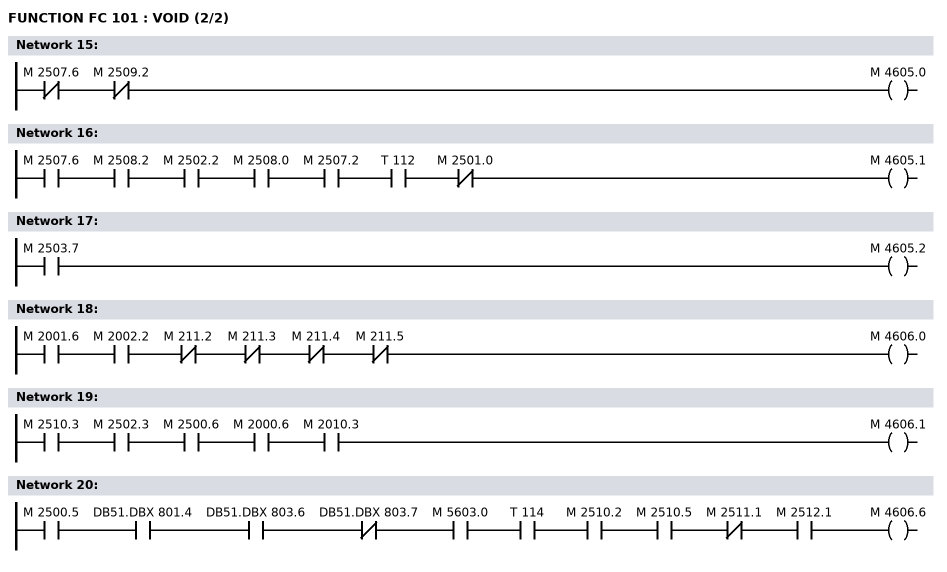

      AN    M   2507.6;
      AN    M   2509.2;
      =     M   4605.0;
NETWORK
TITLE =

      A     M   2507.6;
      A     M   2508.2;
      A     M   2502.2;
      A     M   2508.0;
      A     M   2507.2;
      A     T    112;
      AN    M   2501.0;
      =     M   4605.1;
NETWORK
TITLE =

      A     M   2503.7;
      =     M   4605.2;
NETWORK
TITLE =

      A     M   2001.6;
      A     M   2002.2;
      AN    M    211.2;
      AN    M    211.3;
      AN    M    211.4;
      AN    M    211.5;
      =     M   4606.0;
NETWORK
TITLE =

      A     M   2510.3;
      A     M   2502.3;
      A     M   2500.6;
      A     M   2000.6;
      A     M   2010.3;
      =     M   4606.1;
NETWORK
TITLE =

      A     M   2500.5;
      A     DB51.DBX  801.4;
      A     DB51.DBX  803.6;
      AN    DB51.DBX  803.7;
      A     M   5603.0;
      A     T    114;
      A     M   2510.2;
      A     M   2510.5;
      AN    M   2511.1;
      A     M   2512.1;
      =     M   4606.6;
END_FUNCTION

FUNCTION FC 102 : VOID
TITLE =
VERSION : 0.1

BEGIN
NETWORK
TITLE =운전준비
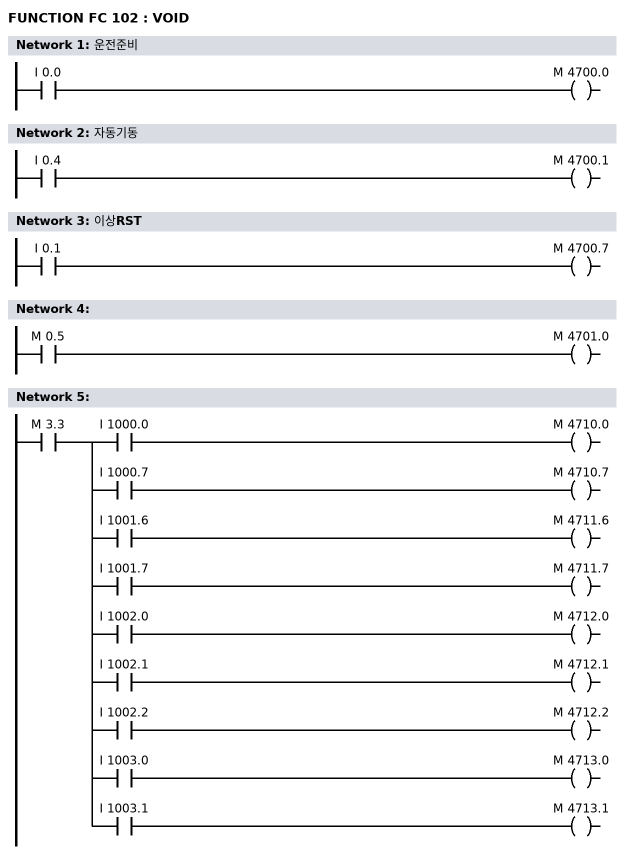

      A     I      0.0;
      =     M   4700.0;
NETWORK
TITLE =자동기동

      A     I      0.4;
      =     M   4700.1;
NETWORK
TITLE =이상RST

      A     I      0.1;
      =     M   4700.7;
NETWORK
TITLE =

      A     M      0.5;
      =     M   4701.0;
NETWORK
TITLE =

      A     M      3.3;
      =     L      0.0;
      A     L      0.0;
      A     I   1000.0;
      =     M   4710.0;
      A     L      0.0;
      A     I   1000.7;
      =     M   4710.7;
      A     L      0.0;
      A     I   1001.6;
      =     M   4711.6;
      A     L      0.0;
      A     I   1001.7;
      =     M   4711.7;
      A     L      0.0;
      A     I   1002.0;
      =     M   4712.0;
      A     L      0.0;
      A     I   1002.1;
      =     M   4712.1;
      A     L      0.0;
      A     I   1002.2;
      =     M   4712.2;
      A     L      0.0;
      A     I   1003.0;
      =     M   4713.0;
      A     L      0.0;
      A     I   1003.1;
      =     M   4713.1;
END_FUNCTION

FUNCTION FC 103 : VOID
TITLE =
VERSION : 0.1

BEGIN
NETWORK
TITLE =
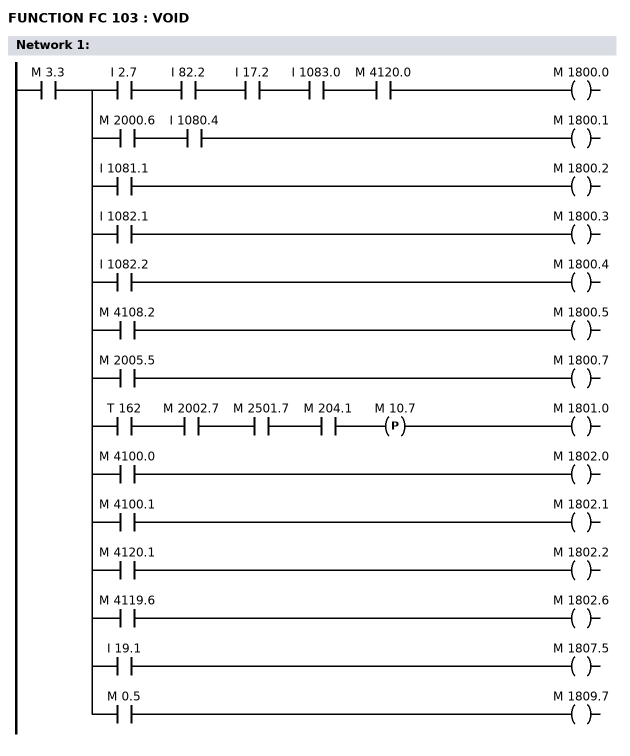

      A     M      3.3;
      =     L      0.0;
      A     L      0.0;
      A     I      2.7;
      A     I     82.2;
      A     I     17.2;
      A     I   1083.0;
      A     M   4120.0;
      =     M   1800.0;
      A     L      0.0;
      A     M   2000.6;
      A     I   1080.4;
      =     M   1800.1;
      A     L      0.0;
      A     I   1081.1;
      =     M   1800.2;
      A     L      0.0;
      A     I   1082.1;
      =     M   1800.3;
      A     L      0.0;
      A     I   1082.2;
      =     M   1800.4;
      A     L      0.0;
      A     M   4108.2;
      =     M   1800.5;
      A     L      0.0;
      A     M   2005.5;
      =     M   1800.7;
      A     L      0.0;
      A     T    162;
      A     M   2002.7;
      A     M   2501.7;
      A     M    204.1;
      FP    M     10.7;
      =     M   1801.0;
      A     L      0.0;
      A     M   4100.0;
      =     M   1802.0;
      A     L      0.0;
      A     M   4100.1;
      =     M   1802.1;
      A     L      0.0;
      A     M   4120.1;
      =     M   1802.2;
      A     L      0.0;
      A     M   4119.6;
      =     M   1802.6;
      A     L      0.0;
      A     I     19.1;
      =     M   1807.5;
      A     L      0.0;
      A     M      0.5;
      =     M   1809.7;
END_FUNCTION

FUNCTION_BLOCK FB 105
TITLE =
VERSION : 0.1


VAR
  S705_RBT1_WELD_OK_PLS : BOOL ;
  S705_RBT1_WELD_NG_PLS : BOOL ;
  S705_RBT1_WELD_PASS_PLS : BOOL ;
  S705_CHECK_SUM_PLS : BOOL ;
  S705_WELD_DATA_MOV_BUFF : BOOL ;
  MW_0_BUFF : ARRAY  [0 .. 59 ] OF WORD ;
  S706_RBT1_WELD_OK_PLS : BOOL ;
  S706_RBT1_WELD_NG_PLS : BOOL ;
  S706_RBT1_WELD_PASS_PLS : BOOL ;
  S706_RBT2_WELD_OK_PLS : BOOL ;
  S706_RBT2_WELD_NG_PLS : BOOL ;
  S706_RBT2_WELD_PASS_PLS : BOOL ;
  S706_RBT3_WELD_OK_PLS : BOOL ;
  S706_RBT3_WELD_NG_PLS : BOOL ;
  S706_RBT3_WELD_PASS_PLS : BOOL ;
  S706_CHECK_SUM_PLS : BOOL ;
  S706_WELD_DATA_MOV_BUFF : BOOL ;
  S711_RBT1_WELD_OK_PLS : BOOL ;
  S711_RBT1_WELD_NG_PLS : BOOL ;
  S711_RBT1_WELD_PASS_PLS : BOOL ;
  S711_CHECK_SUM_PLS : BOOL ;
  S711_WELD_DATA_MOV_BUFF : BOOL ;
  PLS1 : BOOL ;
  PLS2 : BOOL ;
  PLS3 : BOOL ;
  PLS4 : BOOL ;
  PLS5 : BOOL ;
  PLS6 : BOOL ;
END_VAR
VAR_TEMP
  SFC20_RET_VAL : INT ;
END_VAR
BEGIN
NETWORK
TITLE =MES 용접누락 DATA -> #705차종코드(2011) 기준값 버퍼로 전송(LM)
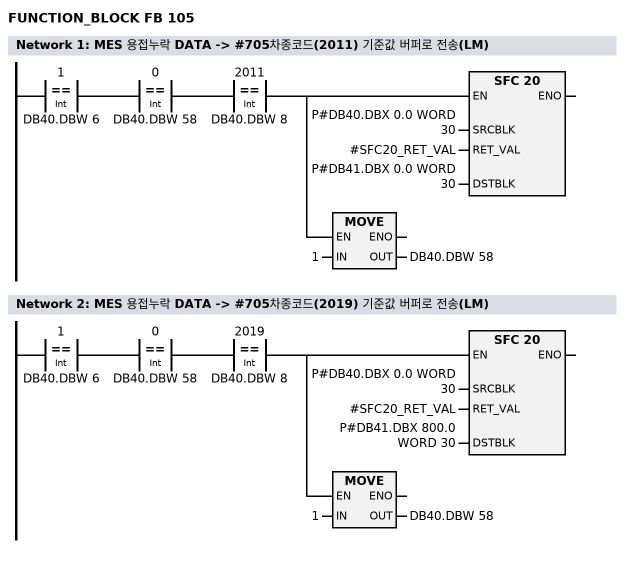

      A(    ;
      L     1;
      L     DB40.DBW    6;
      ==I   ;
      )     ;
      A(    ;
      L     0;
      L     DB40.DBW   58;
      ==I   ;
      )     ;
      A(    ;
      L     2011;
      L     DB40.DBW    8;
      ==I   ;
      )     ;
      =     L      2.0;
      A     L      2.0;
      JNB   _001;
      CALL SFC   20 (
           SRCBLK                   := P#DB40.DBX 0.0 WORD 30,
           RET_VAL                  := #SFC20_RET_VAL,
           DSTBLK                   := P#DB41.DBX 0.0 WORD 30);
_001: NOP   0;
      A     L      2.0;
      JNB   _002;
      L     1;
      T     DB40.DBW   58;
_002: NOP   0;
NETWORK
TITLE =MES 용접누락 DATA -> #705차종코드(2019) 기준값 버퍼로 전송(LM)

      A(    ;
      L     1;
      L     DB40.DBW    6;
      ==I   ;
      )     ;
      A(    ;
      L     0;
      L     DB40.DBW   58;
      ==I   ;
      )     ;
      A(    ;
      L     2019;
      L     DB40.DBW    8;
      ==I   ;
      )     ;
      =     L      2.0;
      A     L      2.0;
      JNB   _003;
      CALL SFC   20 (
           SRCBLK                   := P#DB40.DBX 0.0 WORD 30,
           RET_VAL                  := #SFC20_RET_VAL,
           DSTBLK                   := P#DB41.DBX 800.0 WORD 30);
_003: NOP   0;
      A     L      2.0;
      JNB   _004;
      L     1;
      T     DB40.DBW   58;
_004: NOP   0;
NETWORK
TITLE =#705 RBT1호 용접카운터 INT -> DB로 전송보조

      AN    OV;
      =     L      2.0;
      A     L      2.0;
      A     I   1004.0;
      =     M     11.0;
      A     L      2.0;
      A     I   1004.1;
      =     M     11.1;
      A     L      2.0;
      A     I   1004.2;
      =     M     11.2;
      A     L      2.0;
      A     I   1004.3;
      =     M     11.3;
      A     L      2.0;
      A     I   1004.4;
      =     M     11.4;
      A     L      2.0;
      AN    M      3.3;
      =     L      2.1;
      A     L      2.1;
      A     I   1004.5;
      =     M     11.5;
      A     L      2.1;
      A     I   1004.6;
      =     M     11.6;
      A     L      2.1;
      A     I   1004.7;
      =     M     11.7;
NETWORK
TITLE =#705 RBT1호 용접카운터 INT -> DB로 전송
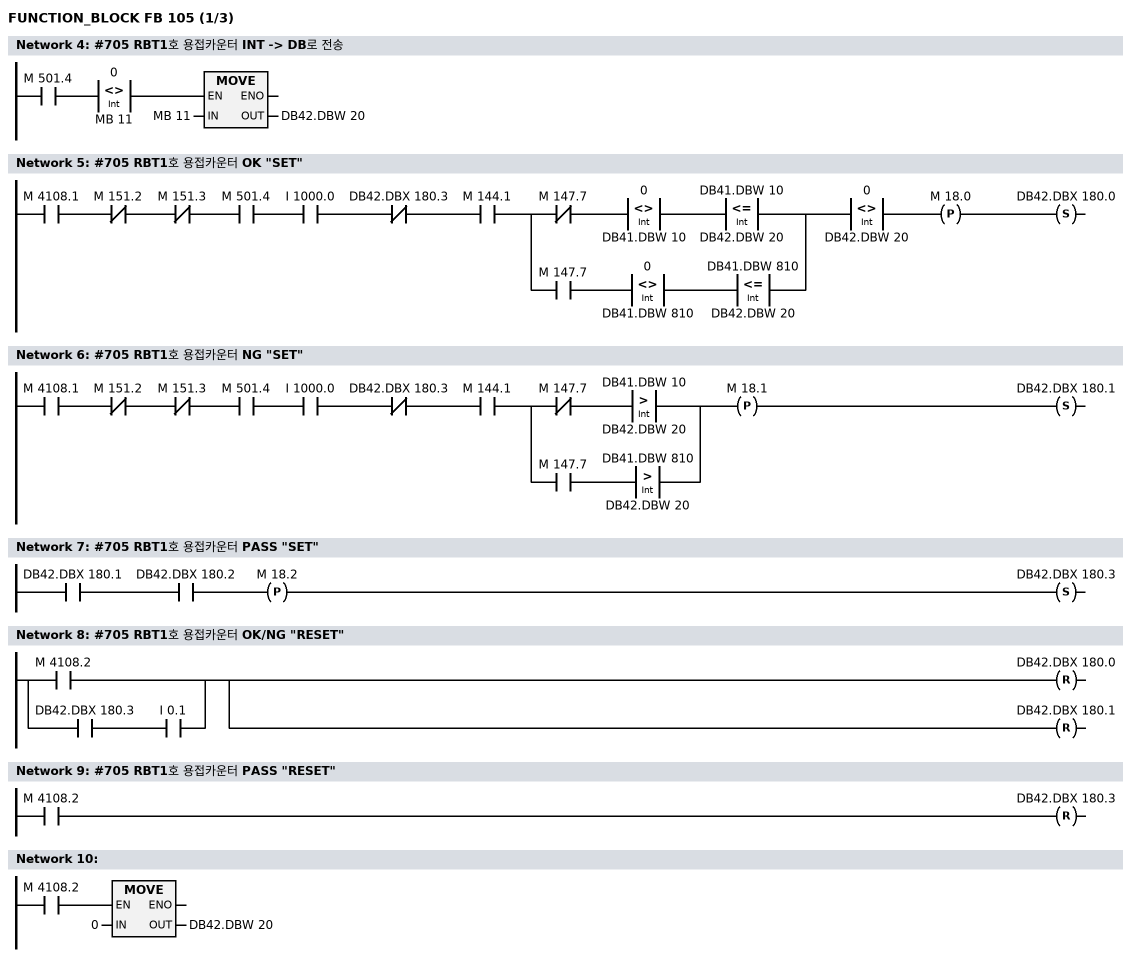

      A     M    501.4;
      A(    ;
      L     0;
      L     MB    11;
      <>I   ;
      )     ;
      JNB   _005;
      L     MB    11;
      T     DB42.DBW   20;
_005: NOP   0;
NETWORK
TITLE =#705 RBT1호 용접카운터 OK "SET"

      A     M   4108.1;
      AN    M    151.2;
      AN    M    151.3;
      A     M    501.4;
      A     I   1000.0;
      AN    DB42.DBX  180.3;
      A     M    144.1;
      A(    ;
      AN    M    147.7;
      A(    ;
      L     0;
      L     DB41.DBW   10;
      <>I   ;
      )     ;
      A(    ;
      L     DB41.DBW   10;
      L     DB42.DBW   20;
      <=I   ;
      )     ;
      O     ;
      A     M    147.7;
      A(    ;
      L     0;
      L     DB41.DBW  810;
      <>I   ;
      )     ;
      A(    ;
      L     DB41.DBW  810;
      L     DB42.DBW   20;
      <=I   ;
      )     ;
      )     ;
      A(    ;
      L     0;
      L     DB42.DBW   20;
      <>I   ;
      )     ;
      FP    M     18.0;
      S     DB42.DBX  180.0;
NETWORK
TITLE =#705 RBT1호 용접카운터 NG "SET"

      A     M   4108.1;
      AN    M    151.2;
      AN    M    151.3;
      A     M    501.4;
      A     I   1000.0;
      AN    DB42.DBX  180.3;
      A     M    144.1;
      A(    ;
      AN    M    147.7;
      A(    ;
      L     DB41.DBW   10;
      L     DB42.DBW   20;
      >I    ;
      )     ;
      O     ;
      A     M    147.7;
      A(    ;
      L     DB41.DBW  810;
      L     DB42.DBW   20;
      >I    ;
      )     ;
      )     ;
      FP    M     18.1;
      S     DB42.DBX  180.1;
NETWORK
TITLE =#705 RBT1호 용접카운터 PASS "SET"

      A     DB42.DBX  180.1;
      A     DB42.DBX  180.2;
      FP    M     18.2;
      S     DB42.DBX  180.3;
NETWORK
TITLE =#705 RBT1호 용접카운터 OK/NG "RESET"

      O     M   4108.2;
      O     ;
      A     DB42.DBX  180.3;
      A     I      0.1;
      R     DB42.DBX  180.0;
      R     DB42.DBX  180.1;
NETWORK
TITLE =#705 RBT1호 용접카운터 PASS "RESET"

      A     M   4108.2;
      R     DB42.DBX  180.3;
NETWORK
TITLE =

      A     M   4108.2;
      JNB   _006;
      L     0;
      T     DB42.DBW   20;
_006: NOP   0;
NETWORK
TITLE =
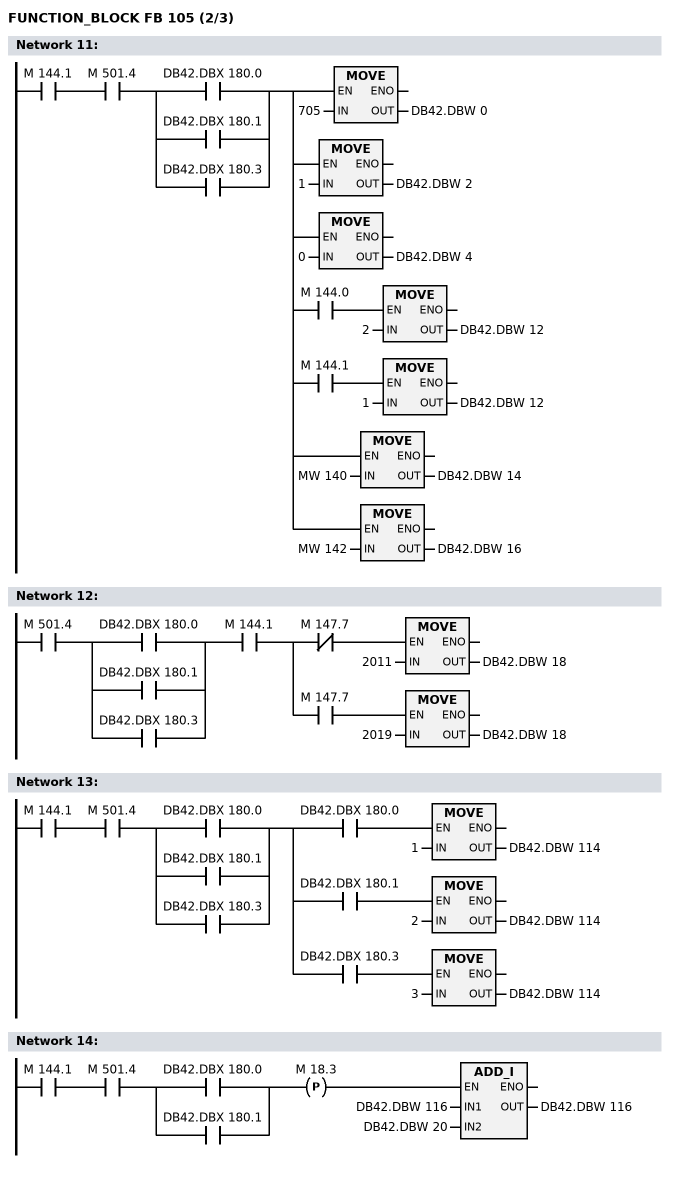

      A     M    144.1;
      A     M    501.4;
      A(    ;
      O     DB42.DBX  180.0;
      O     DB42.DBX  180.1;
      O     DB42.DBX  180.3;
      )     ;
      =     L      2.0;
      A     L      2.0;
      JNB   _007;
      L     705;
      T     DB42.DBW    0;
_007: NOP   0;
      A     L      2.0;
      JNB   _008;
      L     1;
      T     DB42.DBW    2;
_008: NOP   0;
      A     L      2.0;
      JNB   _009;
      L     0;
      T     DB42.DBW    4;
_009: NOP   0;
      A     L      2.0;
      A     M    144.0;
      JNB   _00a;
      L     2;
      T     DB42.DBW   12;
_00a: NOP   0;
      A     L      2.0;
      A     M    144.1;
      JNB   _00b;
      L     1;
      T     DB42.DBW   12;
_00b: NOP   0;
      A     L      2.0;
      JNB   _00c;
      L     MW   140;
      T     DB42.DBW   14;
_00c: NOP   0;
      A     L      2.0;
      JNB   _00d;
      L     MW   142;
      T     DB42.DBW   16;
_00d: NOP   0;
NETWORK
TITLE =

      A     M    501.4;
      A(    ;
      O     DB42.DBX  180.0;
      O     DB42.DBX  180.1;
      O     DB42.DBX  180.3;
      )     ;
      A     M    144.1;
      =     L      2.0;
      A     L      2.0;
      AN    M    147.7;
      JNB   _00e;
      L     2011;
      T     DB42.DBW   18;
_00e: NOP   0;
      A     L      2.0;
      A     M    147.7;
      JNB   _00f;
      L     2019;
      T     DB42.DBW   18;
_00f: NOP   0;
NETWORK
TITLE =

      A     M    144.1;
      A     M    501.4;
      A(    ;
      O     DB42.DBX  180.0;
      O     DB42.DBX  180.1;
      O     DB42.DBX  180.3;
      )     ;
      =     L      2.0;
      A     L      2.0;
      A     DB42.DBX  180.0;
      JNB   _010;
      L     1;
      T     DB42.DBW  114;
_010: NOP   0;
      A     L      2.0;
      A     DB42.DBX  180.1;
      JNB   _011;
      L     2;
      T     DB42.DBW  114;
_011: NOP   0;
      A     L      2.0;
      A     DB42.DBX  180.3;
      JNB   _012;
      L     3;
      T     DB42.DBW  114;
_012: NOP   0;
NETWORK
TITLE =

      A     M    144.1;
      A     M    501.4;
      A(    ;
      O     DB42.DBX  180.0;
      O     DB42.DBX  180.1;
      )     ;
      FP    M     18.3;
      JNB   _013;
      L     DB42.DBW  116;
      L     DB42.DBW   20;
      +I    ;
      T     DB42.DBW  116;
_013: NOP   0;
NETWORK
TITLE =
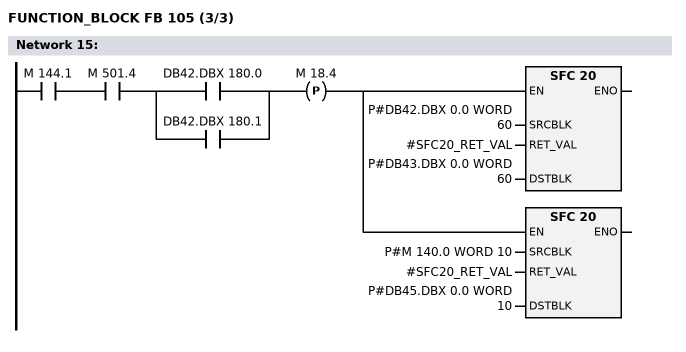

      A     M    144.1;
      A     M    501.4;
      A(    ;
      O     DB42.DBX  180.0;
      O     DB42.DBX  180.1;
      )     ;
      FP    M     18.4;
      =     L      2.0;
      A     L      2.0;
      JNB   _014;
      CALL SFC   20 (
           SRCBLK                   := P#DB42.DBX 0.0 WORD 60,
           RET_VAL                  := #SFC20_RET_VAL,
           DSTBLK                   := P#DB43.DBX 0.0 WORD 60);
_014: NOP   0;
      A     L      2.0;
      JNB   _015;
      CALL SFC   20 (
           SRCBLK                   := P#M 140.0 WORD 10,
           RET_VAL                  := #SFC20_RET_VAL,
           DSTBLK                   := P#DB45.DBX 0.0 WORD 10);
_015: NOP   0;
NETWORK
TITLE =

      A     M   4108.2;
      FP    M     18.5;
      =     L      2.0;
      A(    ;
      A     L      2.0;
      JNB   _016;
      CALL SFC   20 (
           SRCBLK                   := P#DB43.DBX 960.0 WORD 60,
           RET_VAL                  := #SFC20_RET_VAL,
           DSTBLK                   := P#DB43.DBX 1080.0 WORD 60);
_016: A     BR;
      )     ;
      JNB   _017;
      CALL SFC   20 (
           SRCBLK                   := P#DB43.DBX 840.0 WORD 60,
           RET_VAL                  := #SFC20_RET_VAL,
           DSTBLK                   := P#DB43.DBX 960.0 WORD 60);
_017: NOP   0;
      A(    ;
      A     L      2.0;
      JNB   _018;
      CALL SFC   20 (
           SRCBLK                   := P#DB43.DBX 720.0 WORD 60,
           RET_VAL                  := #SFC20_RET_VAL,
           DSTBLK                   := P#DB43.DBX 840.0 WORD 60);
_018: A     BR;
      )     ;
      JNB   _019;
      CALL SFC   20 (
           SRCBLK                   := P#DB43.DBX 600.0 WORD 60,
           RET_VAL                  := #SFC20_RET_VAL,
           DSTBLK                   := P#DB43.DBX 720.0 WORD 60);
_019: NOP   0;
      A(    ;
      A     L      2.0;
      JNB   _01a;
      CALL SFC   20 (
           SRCBLK                   := P#DB43.DBX 480.0 WORD 60,
           RET_VAL                  := #SFC20_RET_VAL,
           DSTBLK                   := P#DB43.DBX 600.0 WORD 60);
_01a: A     BR;
      )     ;
      JNB   _01b;
      CALL SFC   20 (
           SRCBLK                   := P#DB43.DBX 360.0 WORD 60,
           RET_VAL                  := #SFC20_RET_VAL,
           DSTBLK                   := P#DB43.DBX 480.0 WORD 60);
_01b: NOP   0;
      A(    ;
      A     L      2.0;
      JNB   _01c;
      CALL SFC   20 (
           SRCBLK                   := P#DB43.DBX 240.0 WORD 60,
           RET_VAL                  := #SFC20_RET_VAL,
           DSTBLK                   := P#DB43.DBX 360.0 WORD 60);
_01c: A     BR;
      )     ;
      JNB   _01d;
      CALL SFC   20 (
           SRCBLK                   := P#DB43.DBX 120.0 WORD 60,
           RET_VAL                  := #SFC20_RET_VAL,
           DSTBLK                   := P#DB43.DBX 240.0 WORD 60);
_01d: NOP   0;
      A     L      2.0;
      JNB   _01e;
      CALL SFC   20 (
           SRCBLK                   := P#DB43.DBX 0.0 WORD 60,
           RET_VAL                  := #SFC20_RET_VAL,
           DSTBLK                   := P#DB43.DBX 120.0 WORD 60);
_01e: NOP   0;
      A     L      2.0;
      JNB   _01f;
      CALL SFC   21 (
           IN0                      := P#M 40.0 WORD 1,
           RET_VAL                  := #SFC20_RET_VAL,
           OUT1                     := P#DB43.DBX 0.0 WORD 60);
_01f: NOP   0;
      A(    ;
      A     L      2.0;
      JNB   _020;
      CALL SFC   20 (
           SRCBLK                   := P#DB45.DBX 160.0 WORD 10,
           RET_VAL                  := #SFC20_RET_VAL,
           DSTBLK                   := P#DB45.DBX 180.0 WORD 10);
_020: A     BR;
      )     ;
      JNB   _021;
      CALL SFC   20 (
           SRCBLK                   := P#DB45.DBX 140.0 WORD 10,
           RET_VAL                  := #SFC20_RET_VAL,
           DSTBLK                   := P#DB45.DBX 160.0 WORD 10);
_021: NOP   0;
      A(    ;
      A     L      2.0;
      JNB   _022;
      CALL SFC   20 (
           SRCBLK                   := P#DB45.DBX 120.0 WORD 10,
           RET_VAL                  := #SFC20_RET_VAL,
           DSTBLK                   := P#DB45.DBX 140.0 WORD 10);
_022: A     BR;
      )     ;
      JNB   _023;
      CALL SFC   20 (
           SRCBLK                   := P#DB45.DBX 100.0 WORD 10,
           RET_VAL                  := #SFC20_RET_VAL,
           DSTBLK                   := P#DB45.DBX 120.0 WORD 10);
_023: NOP   0;
      A(    ;
      A     L      2.0;
      JNB   _024;
      CALL SFC   20 (
           SRCBLK                   := P#DB45.DBX 80.0 WORD 10,
           RET_VAL                  := #SFC20_RET_VAL,
           DSTBLK                   := P#DB45.DBX 100.0 WORD 10);
_024: A     BR;
      )     ;
      JNB   _025;
      CALL SFC   20 (
           SRCBLK                   := P#DB45.DBX 60.0 WORD 10,
           RET_VAL                  := #SFC20_RET_VAL,
           DSTBLK                   := P#DB45.DBX 80.0 WORD 10);
_025: NOP   0;
      A(    ;
      A     L      2.0;
      JNB   _026;
      CALL SFC   20 (
           SRCBLK                   := P#DB45.DBX 40.0 WORD 10,
           RET_VAL                  := #SFC20_RET_VAL,
           DSTBLK                   := P#DB45.DBX 60.0 WORD 10);
_026: A     BR;
      )     ;
      JNB   _027;
      CALL SFC   20 (
           SRCBLK                   := P#DB45.DBX 20.0 WORD 10,
           RET_VAL                  := #SFC20_RET_VAL,
           DSTBLK                   := P#DB45.DBX 40.0 WORD 10);
_027: NOP   0;
      A     L      2.0;
      JNB   _028;
      CALL SFC   20 (
           SRCBLK                   := P#DB45.DBX 0.0 WORD 10,
           RET_VAL                  := #SFC20_RET_VAL,
           DSTBLK                   := P#DB45.DBX 20.0 WORD 10);
_028: NOP   0;
      A     L      2.0;
      JNB   _029;
      CALL SFC   21 (
           IN0                      := P#M 40.0 WORD 1,
           RET_VAL                  := #SFC20_RET_VAL,
           OUT1                     := P#DB45.DBX 0.0 WORD 10);
_029: NOP   0;
NETWORK
TITLE =
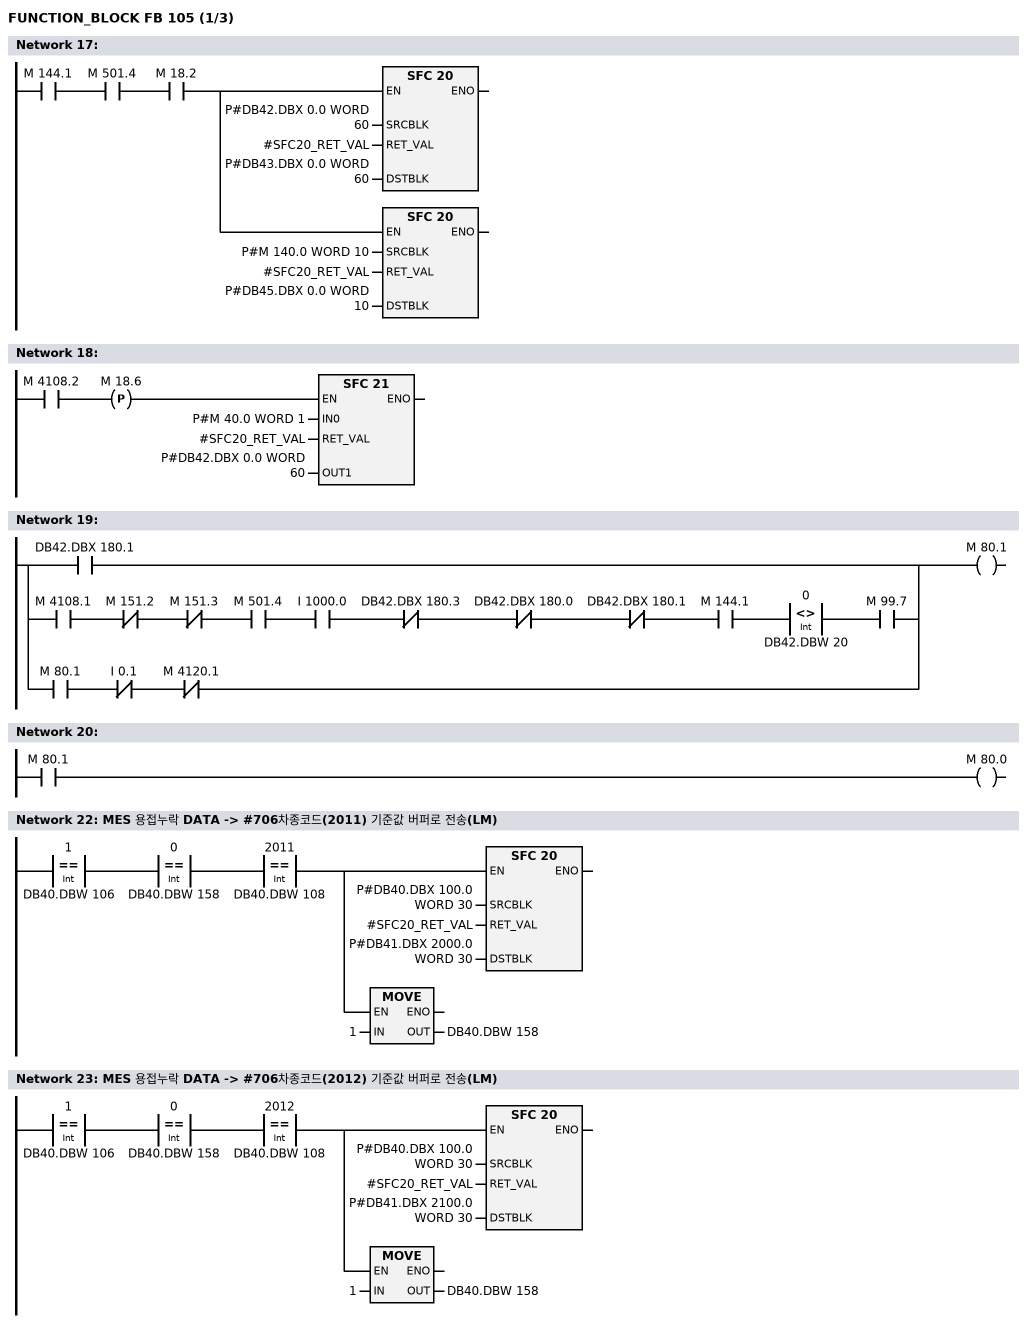

      A     M    144.1;
      A     M    501.4;
      A     M     18.2;
      =     L      2.0;
      A     L      2.0;
      JNB   _02a;
      CALL SFC   20 (
           SRCBLK                   := P#DB42.DBX 0.0 WORD 60,
           RET_VAL                  := #SFC20_RET_VAL,
           DSTBLK                   := P#DB43.DBX 0.0 WORD 60);
_02a: NOP   0;
      A     L      2.0;
      JNB   _02b;
      CALL SFC   20 (
           SRCBLK                   := P#M 140.0 WORD 10,
           RET_VAL                  := #SFC20_RET_VAL,
           DSTBLK                   := P#DB45.DBX 0.0 WORD 10);
_02b: NOP   0;
NETWORK
TITLE =

      A     M   4108.2;
      FP    M     18.6;
      JNB   _02c;
      CALL SFC   21 (
           IN0                      := P#M 40.0 WORD 1,
           RET_VAL                  := #SFC20_RET_VAL,
           OUT1                     := P#DB42.DBX 0.0 WORD 60);
_02c: NOP   0;
NETWORK
TITLE =

      O     DB42.DBX  180.1;
      O     ;
      A     M   4108.1;
      AN    M    151.2;
      AN    M    151.3;
      A     M    501.4;
      A     I   1000.0;
      AN    DB42.DBX  180.3;
      AN    DB42.DBX  180.0;
      AN    DB42.DBX  180.1;
      A     M    144.1;
      A(    ;
      L     0;
      L     DB42.DBW   20;
      <>I   ;
      )     ;
      A     M     99.7;
      O     ;
      A     M     80.1;
      AN    I      0.1;
      AN    M   4120.1;
      =     M     80.1;
NETWORK
TITLE =

      A     M     80.1;
      =     M     80.0;
NETWORK
TITLE =

NETWORK
TITLE =MES 용접누락 DATA -> #706차종코드(2011) 기준값 버퍼로 전송(LM)

      A(    ;
      L     1;
      L     DB40.DBW  106;
      ==I   ;
      )     ;
      A(    ;
      L     0;
      L     DB40.DBW  158;
      ==I   ;
      )     ;
      A(    ;
      L     2011;
      L     DB40.DBW  108;
      ==I   ;
      )     ;
      =     L      2.0;
      A     L      2.0;
      JNB   _02d;
      CALL SFC   20 (
           SRCBLK                   := P#DB40.DBX 100.0 WORD 30,
           RET_VAL                  := #SFC20_RET_VAL,
           DSTBLK                   := P#DB41.DBX 2000.0 WORD 30);
_02d: NOP   0;
      A     L      2.0;
      JNB   _02e;
      L     1;
      T     DB40.DBW  158;
_02e: NOP   0;
NETWORK
TITLE =MES 용접누락 DATA -> #706차종코드(2012) 기준값 버퍼로 전송(LM)

      A(    ;
      L     1;
      L     DB40.DBW  106;
      ==I   ;
      )     ;
      A(    ;
      L     0;
      L     DB40.DBW  158;
      ==I   ;
      )     ;
      A(    ;
      L     2012;
      L     DB40.DBW  108;
      ==I   ;
      )     ;
      =     L      2.0;
      A     L      2.0;
      JNB   _02f;
      CALL SFC   20 (
           SRCBLK                   := P#DB40.DBX 100.0 WORD 30,
           RET_VAL                  := #SFC20_RET_VAL,
           DSTBLK                   := P#DB41.DBX 2100.0 WORD 30);
_02f: NOP   0;
      A     L      2.0;
      JNB   _030;
      L     1;
      T     DB40.DBW  158;
_030: NOP   0;
NETWORK
TITLE =MES 용접누락 DATA -> #706차종코드(2013) 기준값 버퍼로 전송(LM)
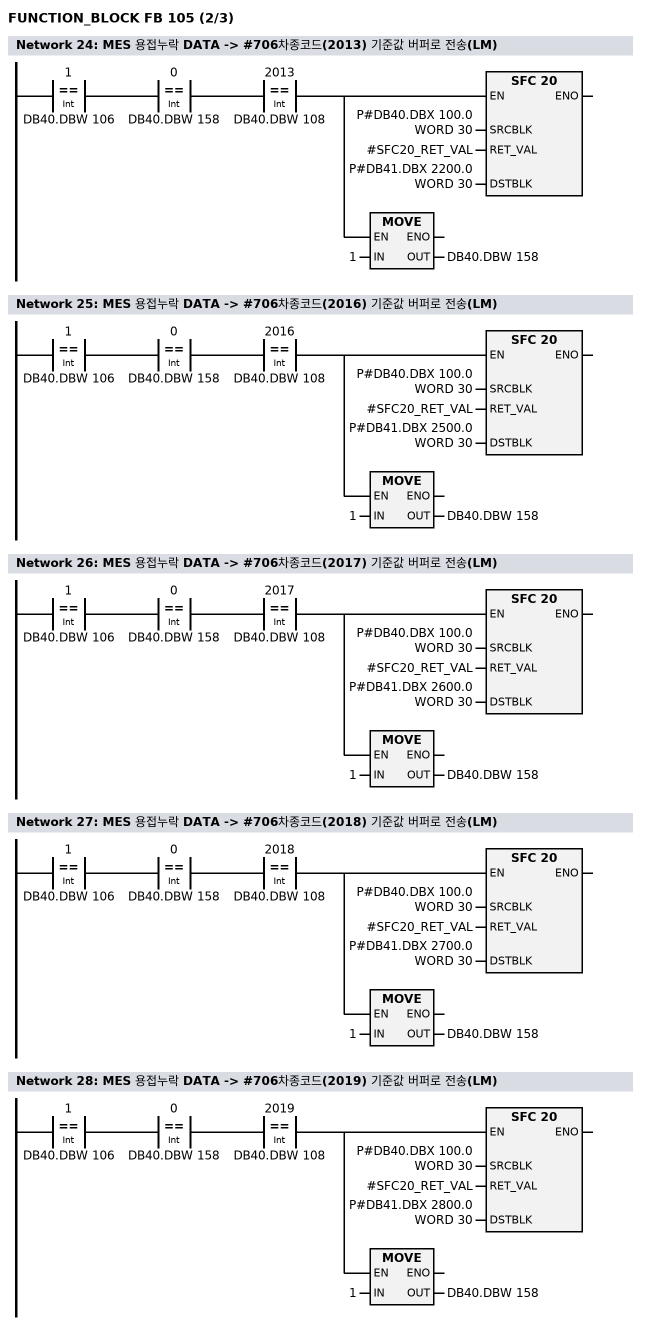

      A(    ;
      L     1;
      L     DB40.DBW  106;
      ==I   ;
      )     ;
      A(    ;
      L     0;
      L     DB40.DBW  158;
      ==I   ;
      )     ;
      A(    ;
      L     2013;
      L     DB40.DBW  108;
      ==I   ;
      )     ;
      =     L      2.0;
      A     L      2.0;
      JNB   _031;
      CALL SFC   20 (
           SRCBLK                   := P#DB40.DBX 100.0 WORD 30,
           RET_VAL                  := #SFC20_RET_VAL,
           DSTBLK                   := P#DB41.DBX 2200.0 WORD 30);
_031: NOP   0;
      A     L      2.0;
      JNB   _032;
      L     1;
      T     DB40.DBW  158;
_032: NOP   0;
NETWORK
TITLE =MES 용접누락 DATA -> #706차종코드(2016) 기준값 버퍼로 전송(LM)

      A(    ;
      L     1;
      L     DB40.DBW  106;
      ==I   ;
      )     ;
      A(    ;
      L     0;
      L     DB40.DBW  158;
      ==I   ;
      )     ;
      A(    ;
      L     2016;
      L     DB40.DBW  108;
      ==I   ;
      )     ;
      =     L      2.0;
      A     L      2.0;
      JNB   _033;
      CALL SFC   20 (
           SRCBLK                   := P#DB40.DBX 100.0 WORD 30,
           RET_VAL                  := #SFC20_RET_VAL,
           DSTBLK                   := P#DB41.DBX 2500.0 WORD 30);
_033: NOP   0;
      A     L      2.0;
      JNB   _034;
      L     1;
      T     DB40.DBW  158;
_034: NOP   0;
NETWORK
TITLE =MES 용접누락 DATA -> #706차종코드(2017) 기준값 버퍼로 전송(LM)

      A(    ;
      L     1;
      L     DB40.DBW  106;
      ==I   ;
      )     ;
      A(    ;
      L     0;
      L     DB40.DBW  158;
      ==I   ;
      )     ;
      A(    ;
      L     2017;
      L     DB40.DBW  108;
      ==I   ;
      )     ;
      =     L      2.0;
      A     L      2.0;
      JNB   _035;
      CALL SFC   20 (
           SRCBLK                   := P#DB40.DBX 100.0 WORD 30,
           RET_VAL                  := #SFC20_RET_VAL,
           DSTBLK                   := P#DB41.DBX 2600.0 WORD 30);
_035: NOP   0;
      A     L      2.0;
      JNB   _036;
      L     1;
      T     DB40.DBW  158;
_036: NOP   0;
NETWORK
TITLE =MES 용접누락 DATA -> #706차종코드(2018) 기준값 버퍼로 전송(LM)

      A(    ;
      L     1;
      L     DB40.DBW  106;
      ==I   ;
      )     ;
      A(    ;
      L     0;
      L     DB40.DBW  158;
      ==I   ;
      )     ;
      A(    ;
      L     2018;
      L     DB40.DBW  108;
      ==I   ;
      )     ;
      =     L      2.0;
      A     L      2.0;
      JNB   _037;
      CALL SFC   20 (
           SRCBLK                   := P#DB40.DBX 100.0 WORD 30,
           RET_VAL                  := #SFC20_RET_VAL,
           DSTBLK                   := P#DB41.DBX 2700.0 WORD 30);
_037: NOP   0;
      A     L      2.0;
      JNB   _038;
      L     1;
      T     DB40.DBW  158;
_038: NOP   0;
NETWORK
TITLE =MES 용접누락 DATA -> #706차종코드(2019) 기준값 버퍼로 전송(LM)

      A(    ;
      L     1;
      L     DB40.DBW  106;
      ==I   ;
      )     ;
      A(    ;
      L     0;
      L     DB40.DBW  158;
      ==I   ;
      )     ;
      A(    ;
      L     2019;
      L     DB40.DBW  108;
      ==I   ;
      )     ;
      =     L      2.0;
      A     L      2.0;
      JNB   _039;
      CALL SFC   20 (
           SRCBLK                   := P#DB40.DBX 100.0 WORD 30,
           RET_VAL                  := #SFC20_RET_VAL,
           DSTBLK                   := P#DB41.DBX 2800.0 WORD 30);
_039: NOP   0;
      A     L      2.0;
      JNB   _03a;
      L     1;
      T     DB40.DBW  158;
_03a: NOP   0;
NETWORK
TITLE =MES 용접누락 DATA -> #706차종코드(2101) 기준값 버퍼로 전송(TL)
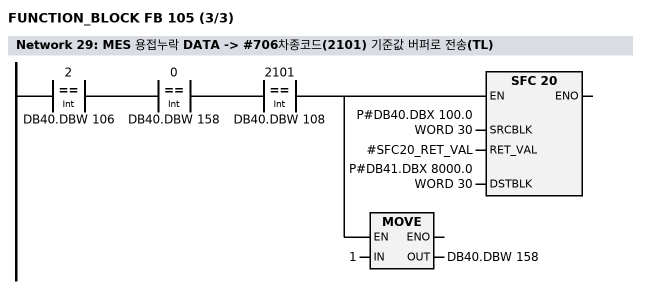

      A(    ;
      L     2;
      L     DB40.DBW  106;
      ==I   ;
      )     ;
      A(    ;
      L     0;
      L     DB40.DBW  158;
      ==I   ;
      )     ;
      A(    ;
      L     2101;
      L     DB40.DBW  108;
      ==I   ;
      )     ;
      =     L      2.0;
      A     L      2.0;
      JNB   _03b;
      CALL SFC   20 (
           SRCBLK                   := P#DB40.DBX 100.0 WORD 30,
           RET_VAL                  := #SFC20_RET_VAL,
           DSTBLK                   := P#DB41.DBX 8000.0 WORD 30);
_03b: NOP   0;
      A     L      2.0;
      JNB   _03c;
      L     1;
      T     DB40.DBW  158;
_03c: NOP   0;
NETWORK
TITLE =#706 RBT1호 용접카운터 INT -> DB로 전송보조

      AN    OV;
      =     L      2.0;
      A     L      2.0;
      A     I   1028.0;
      =     M     12.0;
      A     L      2.0;
      A     I   1028.1;
      =     M     12.1;
      A     L      2.0;
      A     I   1028.2;
      =     M     12.2;
      A     L      2.0;
      A     I   1028.3;
      =     M     12.3;
      A     L      2.0;
      A     I   1028.4;
      =     M     12.4;
      A     L      2.0;
      AN    M      3.3;
      =     L      2.1;
      A     L      2.1;
      A     I   1028.5;
      =     M     12.5;
      A     L      2.1;
      A     I   1028.6;
      =     M     12.6;
      A     L      2.1;
      A     I   1028.7;
      =     M     12.7;
NETWORK
TITLE =#706 RBT1호 용접카운터 INT -> DB로 전송
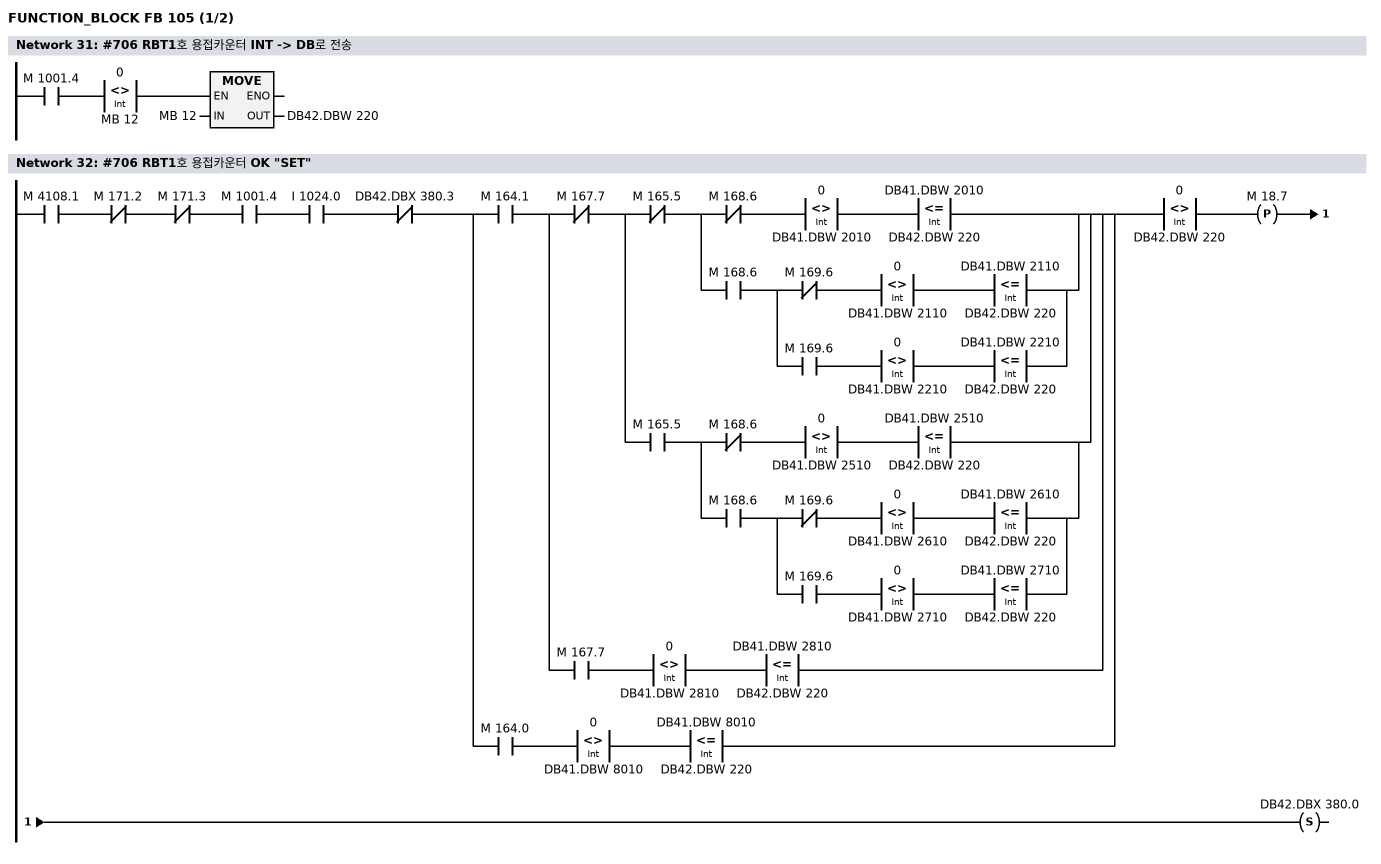

      A     M   1001.4;
      A(    ;
      L     0;
      L     MB    12;
      <>I   ;
      )     ;
      JNB   _03d;
      L     MB    12;
      T     DB42.DBW  220;
_03d: NOP   0;
NETWORK
TITLE =#706 RBT1호 용접카운터 OK "SET"

      A     M   4108.1;
      AN    M    171.2;
      AN    M    171.3;
      A     M   1001.4;
      A     I   1024.0;
      AN    DB42.DBX  380.3;
      A(    ;
      A     M    164.1;
      A(    ;
      AN    M    167.7;
      A(    ;
      AN    M    165.5;
      A(    ;
      AN    M    168.6;
      A(    ;
      L     0;
      L     DB41.DBW 2010;
      <>I   ;
      )     ;
      A(    ;
      L     DB41.DBW 2010;
      L     DB42.DBW  220;
      <=I   ;
      )     ;
      O     ;
      A     M    168.6;
      A(    ;
      AN    M    169.6;
      A(    ;
      L     0;
      L     DB41.DBW 2110;
      <>I   ;
      )     ;
      A(    ;
      L     DB41.DBW 2110;
      L     DB42.DBW  220;
      <=I   ;
      )     ;
      O     ;
      A     M    169.6;
      A(    ;
      L     0;
      L     DB41.DBW 2210;
      <>I   ;
      )     ;
      A(    ;
      L     DB41.DBW 2210;
      L     DB42.DBW  220;
      <=I   ;
      )     ;
      )     ;
      )     ;
      O     ;
      A     M    165.5;
      A(    ;
      AN    M    168.6;
      A(    ;
      L     0;
      L     DB41.DBW 2510;
      <>I   ;
      )     ;
      A(    ;
      L     DB41.DBW 2510;
      L     DB42.DBW  220;
      <=I   ;
      )     ;
      O     ;
      A     M    168.6;
      A(    ;
      AN    M    169.6;
      A(    ;
      L     0;
      L     DB41.DBW 2610;
      <>I   ;
      )     ;
      A(    ;
      L     DB41.DBW 2610;
      L     DB42.DBW  220;
      <=I   ;
      )     ;
      O     ;
      A     M    169.6;
      A(    ;
      L     0;
      L     DB41.DBW 2710;
      <>I   ;
      )     ;
      A(    ;
      L     DB41.DBW 2710;
      L     DB42.DBW  220;
      <=I   ;
      )     ;
      )     ;
      )     ;
      )     ;
      O     ;
      A     M    167.7;
      A(    ;
      L     0;
      L     DB41.DBW 2810;
      <>I   ;
      )     ;
      A(    ;
      L     DB41.DBW 2810;
      L     DB42.DBW  220;
      <=I   ;
      )     ;
      )     ;
      O     ;
      A     M    164.0;
      A(    ;
      L     0;
      L     DB41.DBW 8010;
      <>I   ;
      )     ;
      A(    ;
      L     DB41.DBW 8010;
      L     DB42.DBW  220;
      <=I   ;
      )     ;
      )     ;
      A(    ;
      L     0;
      L     DB42.DBW  220;
      <>I   ;
      )     ;
      FP    M     18.7;
      S     DB42.DBX  380.0;
NETWORK
TITLE =#706 RBT1호 용접카운터 NG "SET"
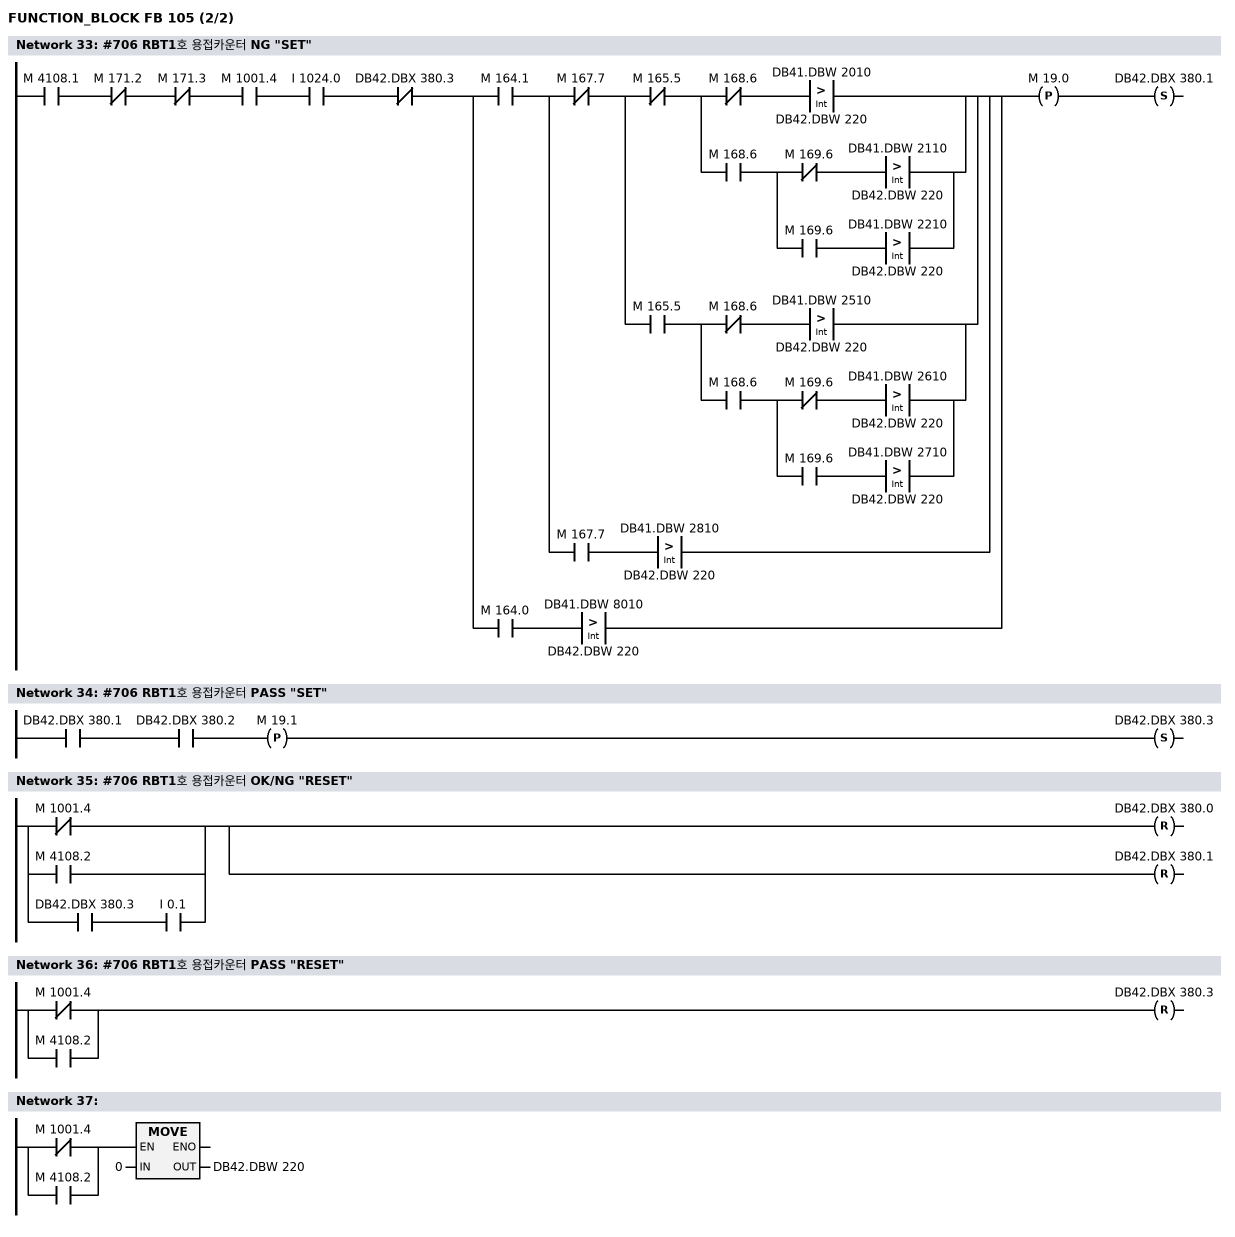

      A     M   4108.1;
      AN    M    171.2;
      AN    M    171.3;
      A     M   1001.4;
      A     I   1024.0;
      AN    DB42.DBX  380.3;
      A(    ;
      A     M    164.1;
      A(    ;
      AN    M    167.7;
      A(    ;
      AN    M    165.5;
      A(    ;
      AN    M    168.6;
      A(    ;
      L     DB41.DBW 2010;
      L     DB42.DBW  220;
      >I    ;
      )     ;
      O     ;
      A     M    168.6;
      A(    ;
      AN    M    169.6;
      A(    ;
      L     DB41.DBW 2110;
      L     DB42.DBW  220;
      >I    ;
      )     ;
      O     ;
      A     M    169.6;
      A(    ;
      L     DB41.DBW 2210;
      L     DB42.DBW  220;
      >I    ;
      )     ;
      )     ;
      )     ;
      O     ;
      A     M    165.5;
      A(    ;
      AN    M    168.6;
      A(    ;
      L     DB41.DBW 2510;
      L     DB42.DBW  220;
      >I    ;
      )     ;
      O     ;
      A     M    168.6;
      A(    ;
      AN    M    169.6;
      A(    ;
      L     DB41.DBW 2610;
      L     DB42.DBW  220;
      >I    ;
      )     ;
      O     ;
      A     M    169.6;
      A(    ;
      L     DB41.DBW 2710;
      L     DB42.DBW  220;
      >I    ;
      )     ;
      )     ;
      )     ;
      )     ;
      O     ;
      A     M    167.7;
      A(    ;
      L     DB41.DBW 2810;
      L     DB42.DBW  220;
      >I    ;
      )     ;
      )     ;
      O     ;
      A     M    164.0;
      A(    ;
      L     DB41.DBW 8010;
      L     DB42.DBW  220;
      >I    ;
      )     ;
      )     ;
      FP    M     19.0;
      S     DB42.DBX  380.1;
NETWORK
TITLE =#706 RBT1호 용접카운터 PASS "SET"

      A     DB42.DBX  380.1;
      A     DB42.DBX  380.2;
      FP    M     19.1;
      S     DB42.DBX  380.3;
NETWORK
TITLE =#706 RBT1호 용접카운터 OK/NG "RESET"

      ON    M   1001.4;
      O     M   4108.2;
      O     ;
      A     DB42.DBX  380.3;
      A     I      0.1;
      R     DB42.DBX  380.0;
      R     DB42.DBX  380.1;
NETWORK
TITLE =#706 RBT1호 용접카운터 PASS "RESET"

      ON    M   1001.4;
      O     M   4108.2;
      R     DB42.DBX  380.3;
NETWORK
TITLE =

      A(    ;
      ON    M   1001.4;
      O     M   4108.2;
      )     ;
      JNB   _03e;
      L     0;
      T     DB42.DBW  220;
_03e: NOP   0;
NETWORK
TITLE =#706 RBT2호 용접카운터 INT -> DB로 전송보조

      AN    OV;
      =     L      2.0;
      A     L      2.0;
      A     I   1036.0;
      =     M     13.0;
      A     L      2.0;
      A     I   1036.1;
      =     M     13.1;
      A     L      2.0;
      A     I   1036.2;
      =     M     13.2;
      A     L      2.0;
      A     I   1036.3;
      =     M     13.3;
      A     L      2.0;
      A     I   1036.4;
      =     M     13.4;
      A     L      2.0;
      AN    M      3.3;
      =     L      2.1;
      A     L      2.1;
      A     I   1036.5;
      =     M     13.5;
      A     L      2.1;
      A     I   1036.6;
      =     M     13.6;
      A     L      2.1;
      A     I   1036.7;
      =     M     13.7;
NETWORK
TITLE =#706 RBT2호 용접카운터 INT -> DB로 전송
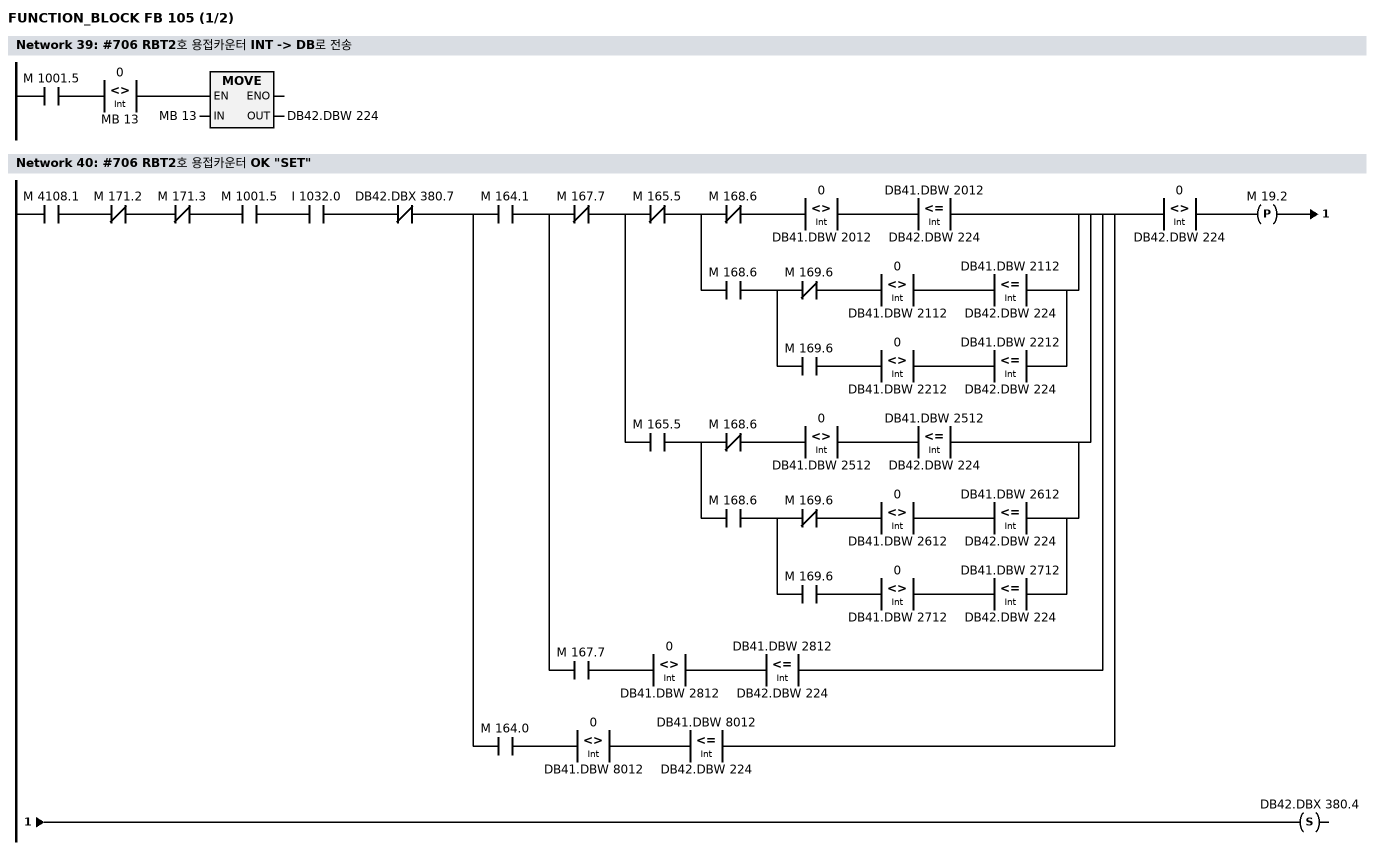

      A     M   1001.5;
      A(    ;
      L     0;
      L     MB    13;
      <>I   ;
      )     ;
      JNB   _03f;
      L     MB    13;
      T     DB42.DBW  224;
_03f: NOP   0;
NETWORK
TITLE =#706 RBT2호 용접카운터 OK "SET"

      A     M   4108.1;
      AN    M    171.2;
      AN    M    171.3;
      A     M   1001.5;
      A     I   1032.0;
      AN    DB42.DBX  380.7;
      A(    ;
      A     M    164.1;
      A(    ;
      AN    M    167.7;
      A(    ;
      AN    M    165.5;
      A(    ;
      AN    M    168.6;
      A(    ;
      L     0;
      L     DB41.DBW 2012;
      <>I   ;
      )     ;
      A(    ;
      L     DB41.DBW 2012;
      L     DB42.DBW  224;
      <=I   ;
      )     ;
      O     ;
      A     M    168.6;
      A(    ;
      AN    M    169.6;
      A(    ;
      L     0;
      L     DB41.DBW 2112;
      <>I   ;
      )     ;
      A(    ;
      L     DB41.DBW 2112;
      L     DB42.DBW  224;
      <=I   ;
      )     ;
      O     ;
      A     M    169.6;
      A(    ;
      L     0;
      L     DB41.DBW 2212;
      <>I   ;
      )     ;
      A(    ;
      L     DB41.DBW 2212;
      L     DB42.DBW  224;
      <=I   ;
      )     ;
      )     ;
      )     ;
      O     ;
      A     M    165.5;
      A(    ;
      AN    M    168.6;
      A(    ;
      L     0;
      L     DB41.DBW 2512;
      <>I   ;
      )     ;
      A(    ;
      L     DB41.DBW 2512;
      L     DB42.DBW  224;
      <=I   ;
      )     ;
      O     ;
      A     M    168.6;
      A(    ;
      AN    M    169.6;
      A(    ;
      L     0;
      L     DB41.DBW 2612;
      <>I   ;
      )     ;
      A(    ;
      L     DB41.DBW 2612;
      L     DB42.DBW  224;
      <=I   ;
      )     ;
      O     ;
      A     M    169.6;
      A(    ;
      L     0;
      L     DB41.DBW 2712;
      <>I   ;
      )     ;
      A(    ;
      L     DB41.DBW 2712;
      L     DB42.DBW  224;
      <=I   ;
      )     ;
      )     ;
      )     ;
      )     ;
      O     ;
      A     M    167.7;
      A(    ;
      L     0;
      L     DB41.DBW 2812;
      <>I   ;
      )     ;
      A(    ;
      L     DB41.DBW 2812;
      L     DB42.DBW  224;
      <=I   ;
      )     ;
      )     ;
      O     ;
      A     M    164.0;
      A(    ;
      L     0;
      L     DB41.DBW 8012;
      <>I   ;
      )     ;
      A(    ;
      L     DB41.DBW 8012;
      L     DB42.DBW  224;
      <=I   ;
      )     ;
      )     ;
      A(    ;
      L     0;
      L     DB42.DBW  224;
      <>I   ;
      )     ;
      FP    M     19.2;
      S     DB42.DBX  380.4;
NETWORK
TITLE =#706 RBT2호 용접카운터 NG "SET"
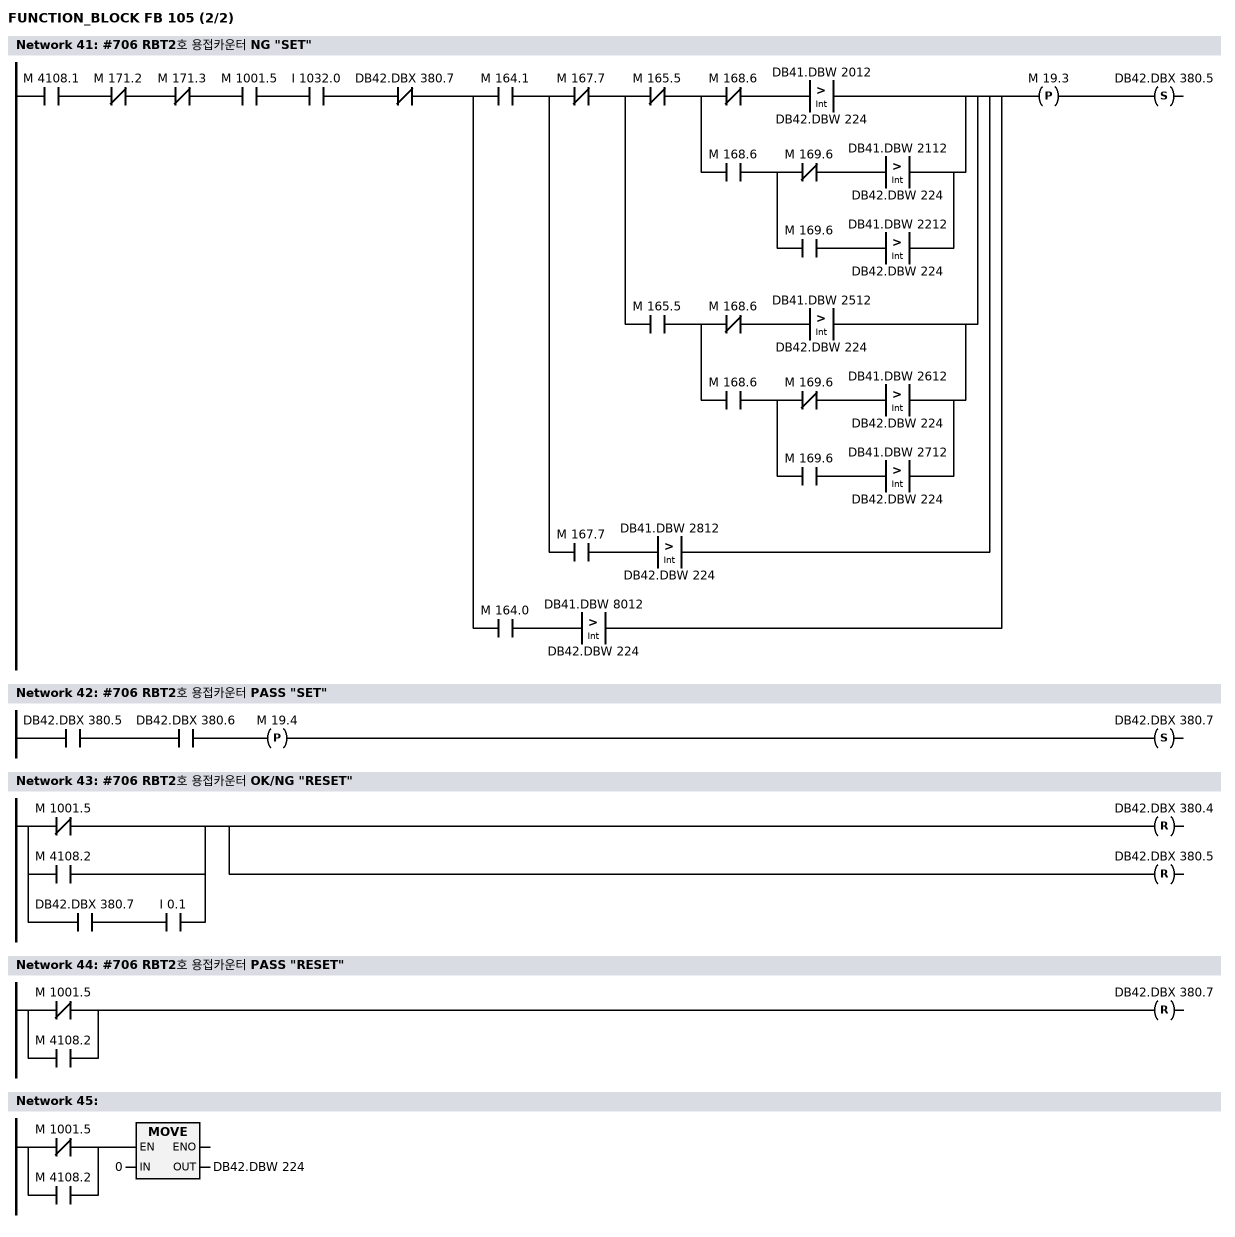

      A     M   4108.1;
      AN    M    171.2;
      AN    M    171.3;
      A     M   1001.5;
      A     I   1032.0;
      AN    DB42.DBX  380.7;
      A(    ;
      A     M    164.1;
      A(    ;
      AN    M    167.7;
      A(    ;
      AN    M    165.5;
      A(    ;
      AN    M    168.6;
      A(    ;
      L     DB41.DBW 2012;
      L     DB42.DBW  224;
      >I    ;
      )     ;
      O     ;
      A     M    168.6;
      A(    ;
      AN    M    169.6;
      A(    ;
      L     DB41.DBW 2112;
      L     DB42.DBW  224;
      >I    ;
      )     ;
      O     ;
      A     M    169.6;
      A(    ;
      L     DB41.DBW 2212;
      L     DB42.DBW  224;
      >I    ;
      )     ;
      )     ;
      )     ;
      O     ;
      A     M    165.5;
      A(    ;
      AN    M    168.6;
      A(    ;
      L     DB41.DBW 2512;
      L     DB42.DBW  224;
      >I    ;
      )     ;
      O     ;
      A     M    168.6;
      A(    ;
      AN    M    169.6;
      A(    ;
      L     DB41.DBW 2612;
      L     DB42.DBW  224;
      >I    ;
      )     ;
      O     ;
      A     M    169.6;
      A(    ;
      L     DB41.DBW 2712;
      L     DB42.DBW  224;
      >I    ;
      )     ;
      )     ;
      )     ;
      )     ;
      O     ;
      A     M    167.7;
      A(    ;
      L     DB41.DBW 2812;
      L     DB42.DBW  224;
      >I    ;
      )     ;
      )     ;
      O     ;
      A     M    164.0;
      A(    ;
      L     DB41.DBW 8012;
      L     DB42.DBW  224;
      >I    ;
      )     ;
      )     ;
      FP    M     19.3;
      S     DB42.DBX  380.5;
NETWORK
TITLE =#706 RBT2호 용접카운터 PASS "SET"

      A     DB42.DBX  380.5;
      A     DB42.DBX  380.6;
      FP    M     19.4;
      S     DB42.DBX  380.7;
NETWORK
TITLE =#706 RBT2호 용접카운터 OK/NG "RESET"

      ON    M   1001.5;
      O     M   4108.2;
      O     ;
      A     DB42.DBX  380.7;
      A     I      0.1;
      R     DB42.DBX  380.4;
      R     DB42.DBX  380.5;
NETWORK
TITLE =#706 RBT2호 용접카운터 PASS "RESET"

      ON    M   1001.5;
      O     M   4108.2;
      R     DB42.DBX  380.7;
NETWORK
TITLE =

      A(    ;
      ON    M   1001.5;
      O     M   4108.2;
      )     ;
      JNB   _040;
      L     0;
      T     DB42.DBW  224;
_040: NOP   0;
NETWORK
TITLE =#706 RBT3호 용접카운터 INT -> DB로 전송보조

      AN    OV;
      =     L      2.0;
      A     L      2.0;
      A     I   1044.0;
      =     M     14.0;
      A     L      2.0;
      A     I   1044.1;
      =     M     14.1;
      A     L      2.0;
      A     I   1044.2;
      =     M     14.2;
      A     L      2.0;
      A     I   1044.3;
      =     M     14.3;
      A     L      2.0;
      A     I   1044.4;
      =     M     14.4;
      A     L      2.0;
      AN    M      3.3;
      =     L      2.1;
      A     L      2.1;
      A     I   1044.5;
      =     M     14.5;
      A     L      2.1;
      A     I   1044.6;
      =     M     14.6;
      A     L      2.1;
      A     I   1044.7;
      =     M     14.7;
NETWORK
TITLE =#706 RBT3호 용접카운터 INT -> DB로 전송
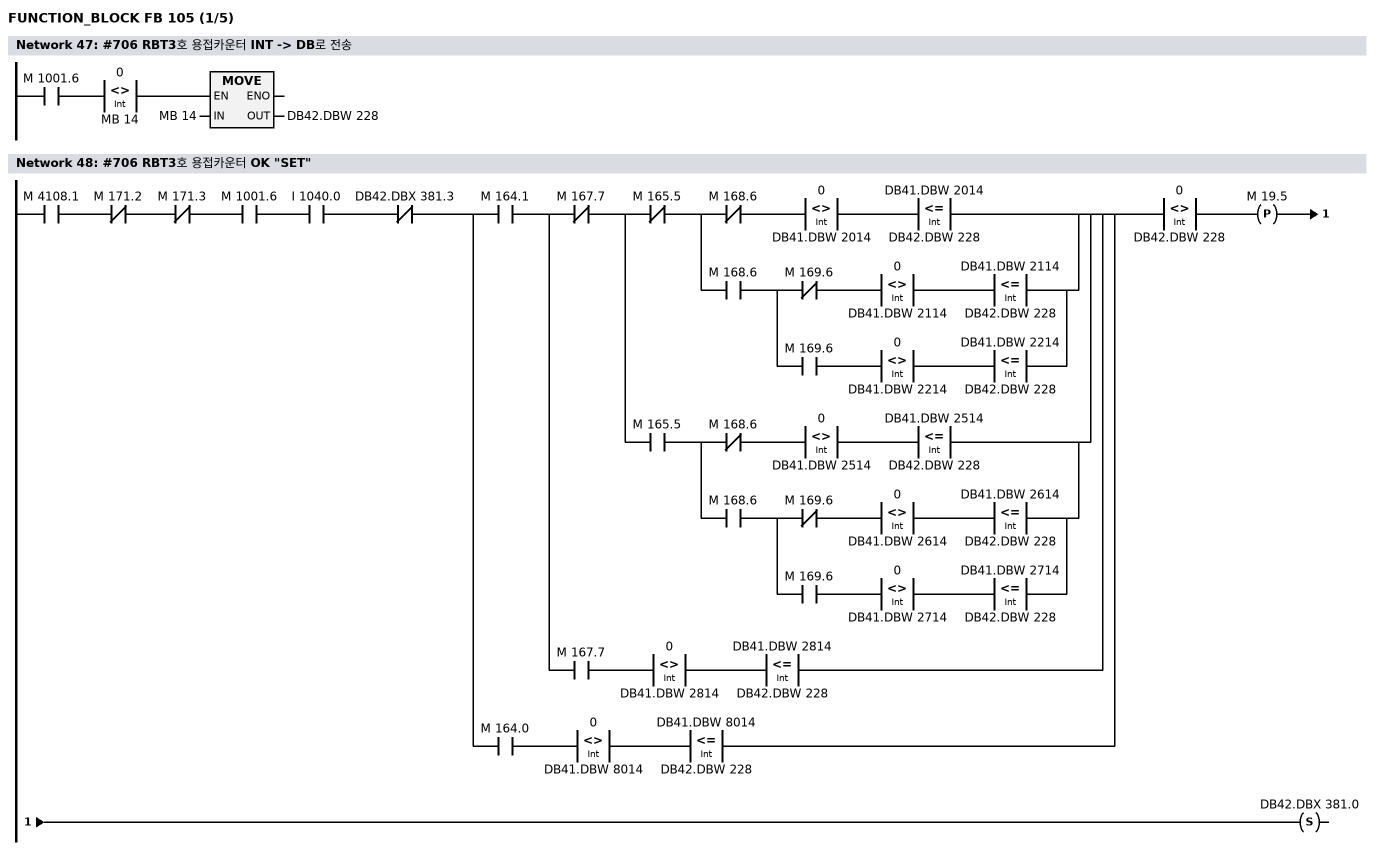

      A     M   1001.6;
      A(    ;
      L     0;
      L     MB    14;
      <>I   ;
      )     ;
      JNB   _041;
      L     MB    14;
      T     DB42.DBW  228;
_041: NOP   0;
NETWORK
TITLE =#706 RBT3호 용접카운터 OK "SET"

      A     M   4108.1;
      AN    M    171.2;
      AN    M    171.3;
      A     M   1001.6;
      A     I   1040.0;
      AN    DB42.DBX  381.3;
      A(    ;
      A     M    164.1;
      A(    ;
      AN    M    167.7;
      A(    ;
      AN    M    165.5;
      A(    ;
      AN    M    168.6;
      A(    ;
      L     0;
      L     DB41.DBW 2014;
      <>I   ;
      )     ;
      A(    ;
      L     DB41.DBW 2014;
      L     DB42.DBW  228;
      <=I   ;
      )     ;
      O     ;
      A     M    168.6;
      A(    ;
      AN    M    169.6;
      A(    ;
      L     0;
      L     DB41.DBW 2114;
      <>I   ;
      )     ;
      A(    ;
      L     DB41.DBW 2114;
      L     DB42.DBW  228;
      <=I   ;
      )     ;
      O     ;
      A     M    169.6;
      A(    ;
      L     0;
      L     DB41.DBW 2214;
      <>I   ;
      )     ;
      A(    ;
      L     DB41.DBW 2214;
      L     DB42.DBW  228;
      <=I   ;
      )     ;
      )     ;
      )     ;
      O     ;
      A     M    165.5;
      A(    ;
      AN    M    168.6;
      A(    ;
      L     0;
      L     DB41.DBW 2514;
      <>I   ;
      )     ;
      A(    ;
      L     DB41.DBW 2514;
      L     DB42.DBW  228;
      <=I   ;
      )     ;
      O     ;
      A     M    168.6;
      A(    ;
      AN    M    169.6;
      A(    ;
      L     0;
      L     DB41.DBW 2614;
      <>I   ;
      )     ;
      A(    ;
      L     DB41.DBW 2614;
      L     DB42.DBW  228;
      <=I   ;
      )     ;
      O     ;
      A     M    169.6;
      A(    ;
      L     0;
      L     DB41.DBW 2714;
      <>I   ;
      )     ;
      A(    ;
      L     DB41.DBW 2714;
      L     DB42.DBW  228;
      <=I   ;
      )     ;
      )     ;
      )     ;
      )     ;
      O     ;
      A     M    167.7;
      A(    ;
      L     0;
      L     DB41.DBW 2814;
      <>I   ;
      )     ;
      A(    ;
      L     DB41.DBW 2814;
      L     DB42.DBW  228;
      <=I   ;
      )     ;
      )     ;
      O     ;
      A     M    164.0;
      A(    ;
      L     0;
      L     DB41.DBW 8014;
      <>I   ;
      )     ;
      A(    ;
      L     DB41.DBW 8014;
      L     DB42.DBW  228;
      <=I   ;
      )     ;
      )     ;
      A(    ;
      L     0;
      L     DB42.DBW  228;
      <>I   ;
      )     ;
      FP    M     19.5;
      S     DB42.DBX  381.0;
NETWORK
TITLE =#706 RBT3호 용접카운터 NG "SET"
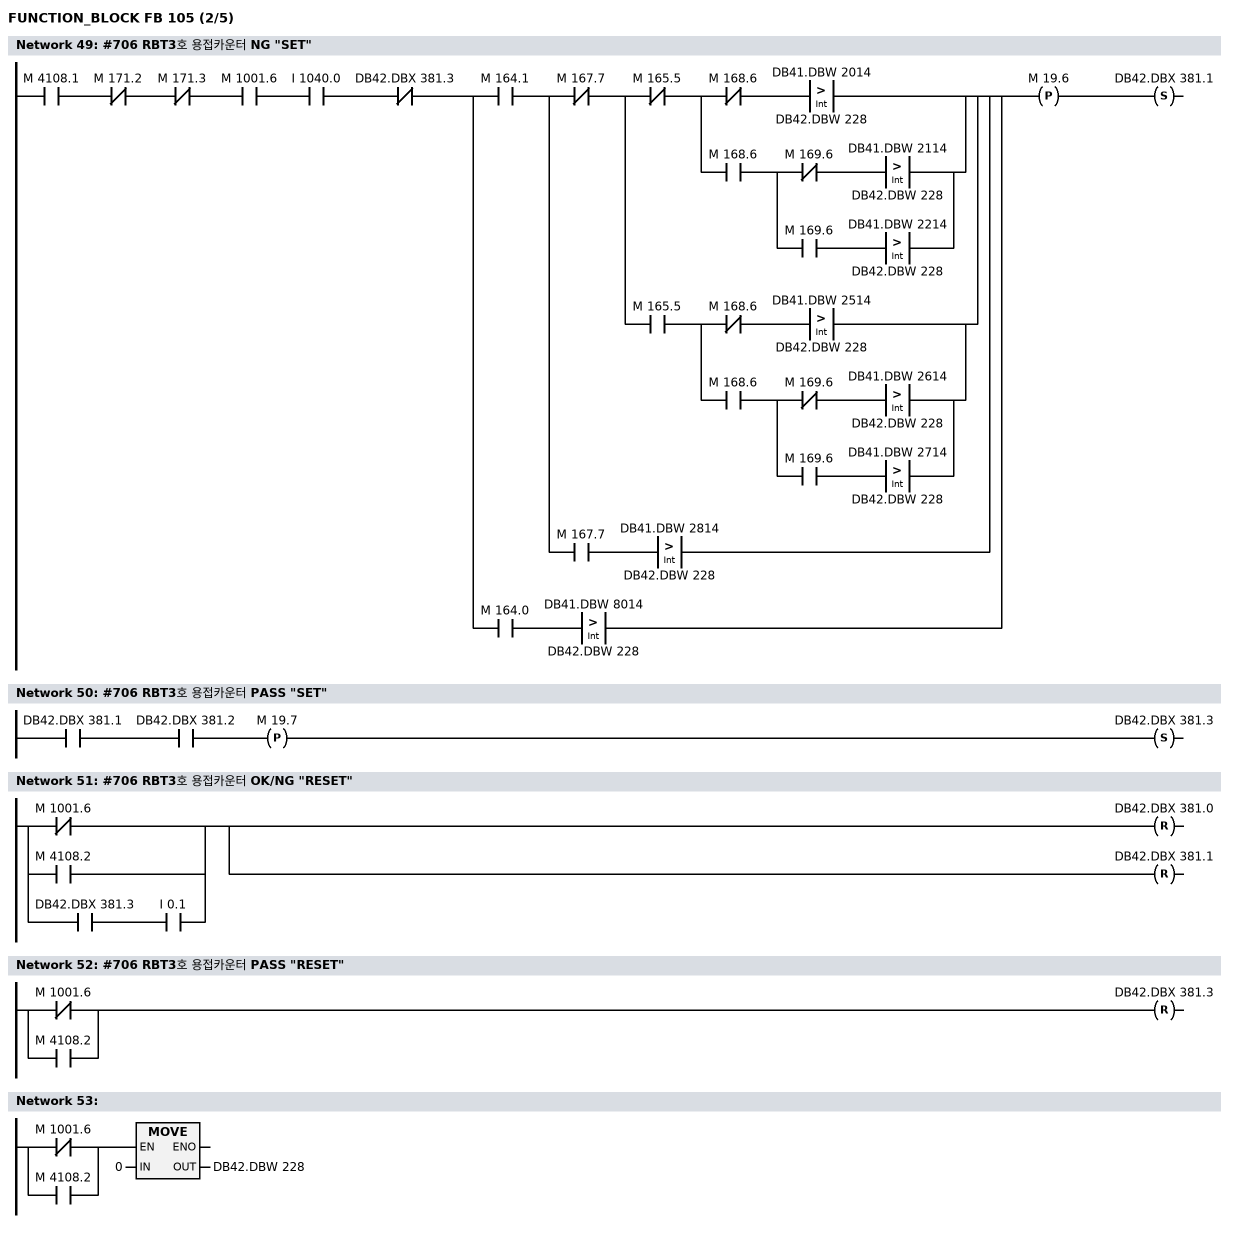

      A     M   4108.1;
      AN    M    171.2;
      AN    M    171.3;
      A     M   1001.6;
      A     I   1040.0;
      AN    DB42.DBX  381.3;
      A(    ;
      A     M    164.1;
      A(    ;
      AN    M    167.7;
      A(    ;
      AN    M    165.5;
      A(    ;
      AN    M    168.6;
      A(    ;
      L     DB41.DBW 2014;
      L     DB42.DBW  228;
      >I    ;
      )     ;
      O     ;
      A     M    168.6;
      A(    ;
      AN    M    169.6;
      A(    ;
      L     DB41.DBW 2114;
      L     DB42.DBW  228;
      >I    ;
      )     ;
      O     ;
      A     M    169.6;
      A(    ;
      L     DB41.DBW 2214;
      L     DB42.DBW  228;
      >I    ;
      )     ;
      )     ;
      )     ;
      O     ;
      A     M    165.5;
      A(    ;
      AN    M    168.6;
      A(    ;
      L     DB41.DBW 2514;
      L     DB42.DBW  228;
      >I    ;
      )     ;
      O     ;
      A     M    168.6;
      A(    ;
      AN    M    169.6;
      A(    ;
      L     DB41.DBW 2614;
      L     DB42.DBW  228;
      >I    ;
      )     ;
      O     ;
      A     M    169.6;
      A(    ;
      L     DB41.DBW 2714;
      L     DB42.DBW  228;
      >I    ;
      )     ;
      )     ;
      )     ;
      )     ;
      O     ;
      A     M    167.7;
      A(    ;
      L     DB41.DBW 2814;
      L     DB42.DBW  228;
      >I    ;
      )     ;
      )     ;
      O     ;
      A     M    164.0;
      A(    ;
      L     DB41.DBW 8014;
      L     DB42.DBW  228;
      >I    ;
      )     ;
      )     ;
      FP    M     19.6;
      S     DB42.DBX  381.1;
NETWORK
TITLE =#706 RBT3호 용접카운터 PASS "SET"

      A     DB42.DBX  381.1;
      A     DB42.DBX  381.2;
      FP    M     19.7;
      S     DB42.DBX  381.3;
NETWORK
TITLE =#706 RBT3호 용접카운터 OK/NG "RESET"

      ON    M   1001.6;
      O     M   4108.2;
      O     ;
      A     DB42.DBX  381.3;
      A     I      0.1;
      R     DB42.DBX  381.0;
      R     DB42.DBX  381.1;
NETWORK
TITLE =#706 RBT3호 용접카운터 PASS "RESET"

      ON    M   1001.6;
      O     M   4108.2;
      R     DB42.DBX  381.3;
NETWORK
TITLE =

      A(    ;
      ON    M   1001.6;
      O     M   4108.2;
      )     ;
      JNB   _042;
      L     0;
      T     DB42.DBW  228;
_042: NOP   0;
NETWORK
TITLE =#706 용접DATA 관련(공정 및 차종정보)
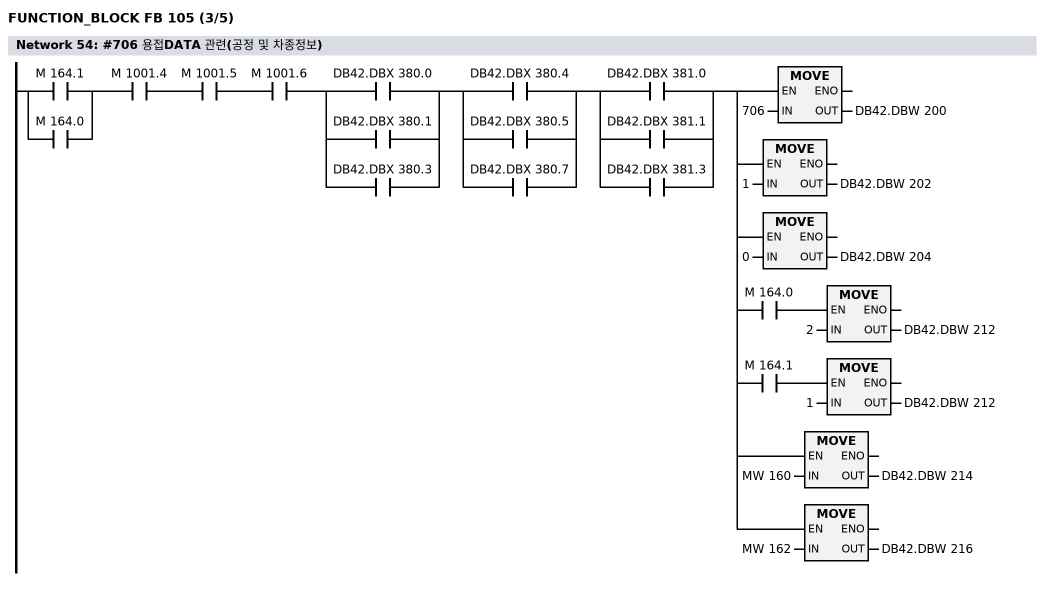

      A(    ;
      O     M    164.1;
      O     M    164.0;
      )     ;
      A     M   1001.4;
      A     M   1001.5;
      A     M   1001.6;
      A(    ;
      O     DB42.DBX  380.0;
      O     DB42.DBX  380.1;
      O     DB42.DBX  380.3;
      )     ;
      A(    ;
      O     DB42.DBX  380.4;
      O     DB42.DBX  380.5;
      O     DB42.DBX  380.7;
      )     ;
      A(    ;
      O     DB42.DBX  381.0;
      O     DB42.DBX  381.1;
      O     DB42.DBX  381.3;
      )     ;
      =     L      2.0;
      A     L      2.0;
      JNB   _043;
      L     706;
      T     DB42.DBW  200;
_043: NOP   0;
      A     L      2.0;
      JNB   _044;
      L     1;
      T     DB42.DBW  202;
_044: NOP   0;
      A     L      2.0;
      JNB   _045;
      L     0;
      T     DB42.DBW  204;
_045: NOP   0;
      A     L      2.0;
      A     M    164.0;
      JNB   _046;
      L     2;
      T     DB42.DBW  212;
_046: NOP   0;
      A     L      2.0;
      A     M    164.1;
      JNB   _047;
      L     1;
      T     DB42.DBW  212;
_047: NOP   0;
      A     L      2.0;
      JNB   _048;
      L     MW   160;
      T     DB42.DBW  214;
_048: NOP   0;
      A     L      2.0;
      JNB   _049;
      L     MW   162;
      T     DB42.DBW  216;
_049: NOP   0;
NETWORK
TITLE =#706 용접DATA 관련(용접 차종CODE)
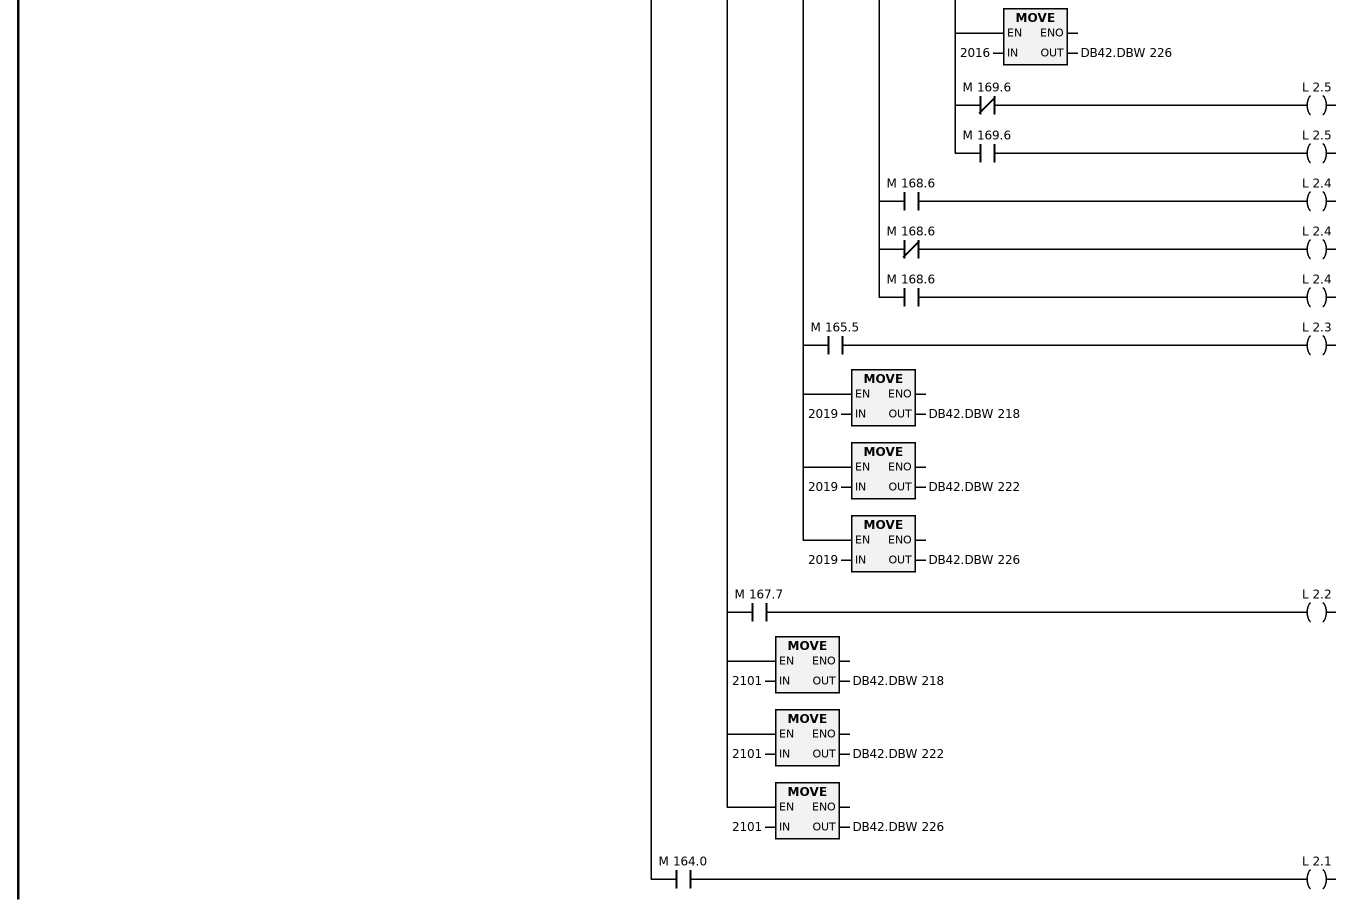

      A     M   1001.4;
      A     M   1001.5;
      A     M   1001.6;
      A(    ;
      O     DB42.DBX  380.0;
      O     DB42.DBX  380.1;
      O     DB42.DBX  380.3;
      )     ;
      A(    ;
      O     DB42.DBX  380.4;
      O     DB42.DBX  380.5;
      O     DB42.DBX  380.7;
      )     ;
      A(    ;
      O     DB42.DBX  381.0;
      O     DB42.DBX  381.1;
      O     DB42.DBX  381.3;
      )     ;
      =     L      2.0;
      A     L      2.0;
      A     M    164.1;
      =     L      2.1;
      A     L      2.1;
      AN    M    167.7;
      =     L      2.2;
      A     L      2.2;
      AN    M    165.5;
      =     L      2.3;
      A     L      2.3;
      AN    M    168.6;
      =     L      2.4;
      A     L      2.4;
      JNB   _04a;
      L     2011;
      T     DB42.DBW  218;
_04a: NOP   0;
      A     L      2.4;
      JNB   _04b;
      L     2011;
      T     DB42.DBW  222;
_04b: NOP   0;
      A     L      2.4;
      JNB   _04c;
      L     2011;
      T     DB42.DBW  226;
_04c: NOP   0;
      A     L      2.3;
      A     M    168.6;
      =     L      2.4;
      A     L      2.4;
      AN    M    169.6;
      =     L      2.5;
      A     L      2.5;
      JNB   _04d;
      L     2012;
      T     DB42.DBW  218;
_04d: NOP   0;
      A     L      2.5;
      JNB   _04e;
      L     2012;
      T     DB42.DBW  222;
_04e: NOP   0;
      A     L      2.5;
      JNB   _04f;
      L     2012;
      T     DB42.DBW  226;
_04f: NOP   0;
      A     L      2.4;
      A     M    169.6;
      =     L      2.5;
      A     L      2.5;
      JNB   _050;
      L     2013;
      T     DB42.DBW  218;
_050: NOP   0;
      A     L      2.5;
      JNB   _051;
      L     2013;
      T     DB42.DBW  222;
_051: NOP   0;
      A     L      2.5;
      JNB   _052;
      L     2013;
      T     DB42.DBW  226;
_052: NOP   0;
      A     L      2.2;
      A     M    165.5;
      =     L      2.3;
      A     L      2.3;
      AN    M    168.6;
      =     L      2.4;
      A     L      2.4;
      JNB   _053;
      L     2016;
      T     DB42.DBW  218;
_053: NOP   0;
      A     L      2.4;
      JNB   _054;
      L     2016;
      T     DB42.DBW  222;
_054: NOP   0;
      A     L      2.4;
      JNB   _055;
      L     2016;
      T     DB42.DBW  226;
_055: NOP   0;
      A     L      2.3;
      A     M    168.6;
      =     L      2.4;
      A     L      2.4;
      AN    M    169.6;
      =     L      2.5;
      A     L      2.5;
      JNB   _056;
      L     2017;
      T     DB42.DBW  218;
_056: NOP   0;
      A     L      2.5;
      JNB   _057;
      L     2017;
      T     DB42.DBW  222;
_057: NOP   0;
      A     L      2.5;
      JNB   _058;
      L     2017;
      T     DB42.DBW  226;
_058: NOP   0;
      A     L      2.4;
      A     M    169.6;
      =     L      2.5;
      A     L      2.5;
      JNB   _059;
      L     2018;
      T     DB42.DBW  218;
_059: NOP   0;
      A     L      2.5;
      JNB   _05a;
      L     2018;
      T     DB42.DBW  222;
_05a: NOP   0;
      A     L      2.5;
      JNB   _05b;
      L     2018;
      T     DB42.DBW  226;
_05b: NOP   0;
      A     L      2.1;
      A     M    167.7;
      =     L      2.2;
      A     L      2.2;
      JNB   _05c;
      L     2019;
      T     DB42.DBW  218;
_05c: NOP   0;
      A     L      2.2;
      JNB   _05d;
      L     2019;
      T     DB42.DBW  222;
_05d: NOP   0;
      A     L      2.2;
      JNB   _05e;
      L     2019;
      T     DB42.DBW  226;
_05e: NOP   0;
      A     L      2.0;
      A     M    164.0;
      =     L      2.1;
      A     L      2.1;
      JNB   _05f;
      L     2101;
      T     DB42.DBW  218;
_05f: NOP   0;
      A     L      2.1;
      JNB   _060;
      L     2101;
      T     DB42.DBW  222;
_060: NOP   0;
      A     L      2.1;
      JNB   _061;
      L     2101;
      T     DB42.DBW  226;
_061: NOP   0;
NETWORK
TITLE =#706 용접DATA 관련(용접결과)
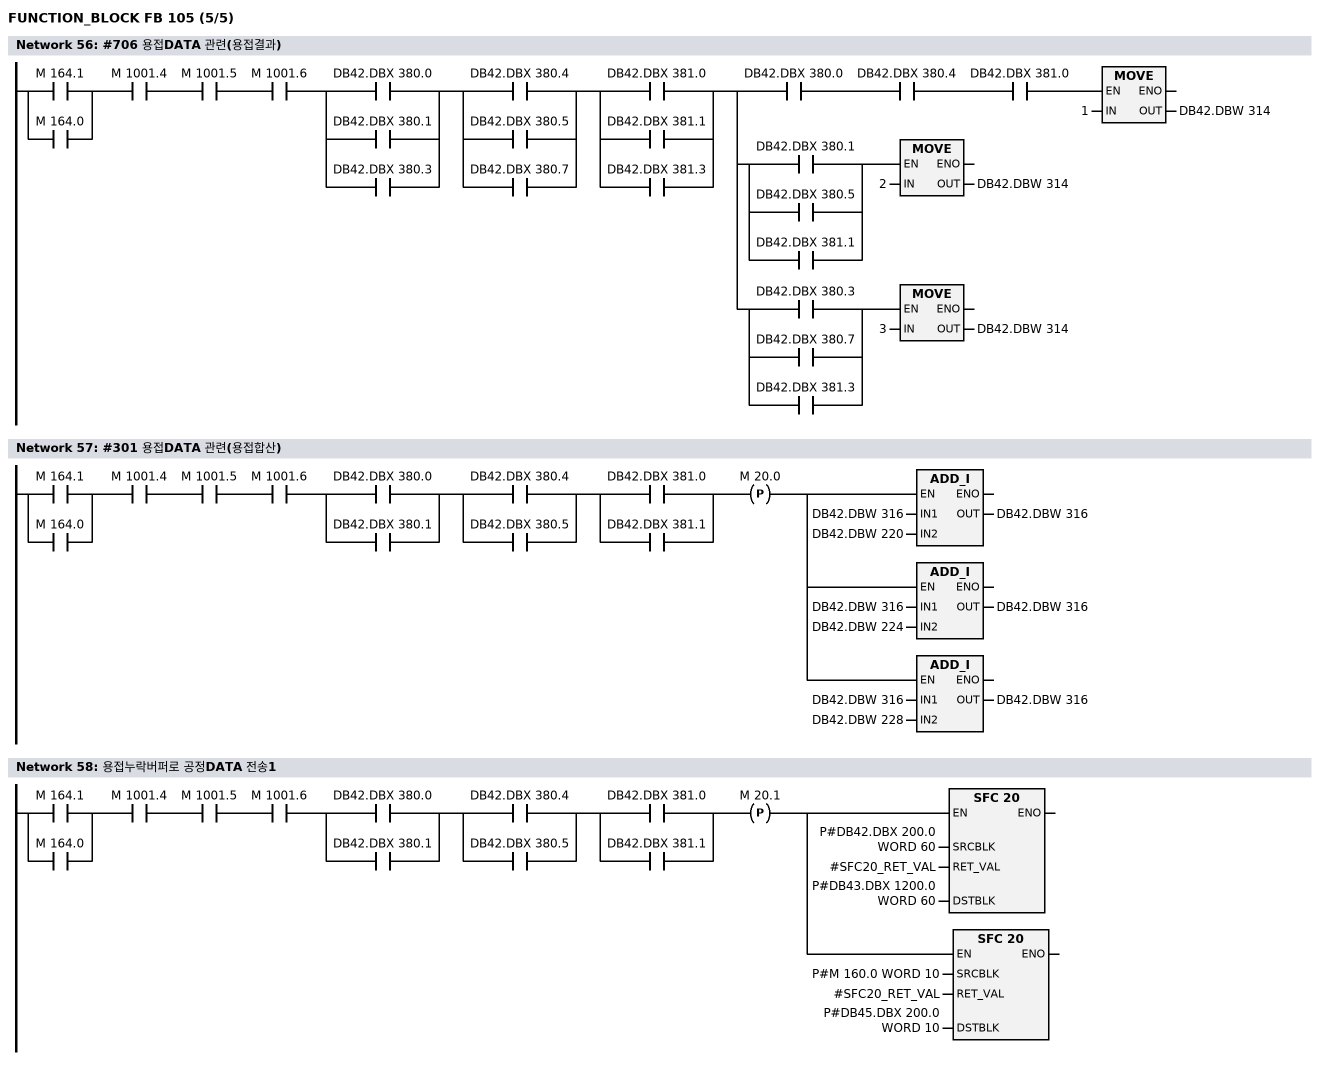

      A(    ;
      O     M    164.1;
      O     M    164.0;
      )     ;
      A     M   1001.4;
      A     M   1001.5;
      A     M   1001.6;
      A(    ;
      O     DB42.DBX  380.0;
      O     DB42.DBX  380.1;
      O     DB42.DBX  380.3;
      )     ;
      A(    ;
      O     DB42.DBX  380.4;
      O     DB42.DBX  380.5;
      O     DB42.DBX  380.7;
      )     ;
      A(    ;
      O     DB42.DBX  381.0;
      O     DB42.DBX  381.1;
      O     DB42.DBX  381.3;
      )     ;
      =     L      2.0;
      A     L      2.0;
      A     DB42.DBX  380.0;
      A     DB42.DBX  380.4;
      A     DB42.DBX  381.0;
      JNB   _062;
      L     1;
      T     DB42.DBW  314;
_062: NOP   0;
      A     L      2.0;
      A(    ;
      O     DB42.DBX  380.1;
      O     DB42.DBX  380.5;
      O     DB42.DBX  381.1;
      )     ;
      JNB   _063;
      L     2;
      T     DB42.DBW  314;
_063: NOP   0;
      A     L      2.0;
      A(    ;
      O     DB42.DBX  380.3;
      O     DB42.DBX  380.7;
      O     DB42.DBX  381.3;
      )     ;
      JNB   _064;
      L     3;
      T     DB42.DBW  314;
_064: NOP   0;
NETWORK
TITLE =#301 용접DATA 관련(용접합산)

      A(    ;
      O     M    164.1;
      O     M    164.0;
      )     ;
      A     M   1001.4;
      A     M   1001.5;
      A     M   1001.6;
      A(    ;
      O     DB42.DBX  380.0;
      O     DB42.DBX  380.1;
      )     ;
      A(    ;
      O     DB42.DBX  380.4;
      O     DB42.DBX  380.5;
      )     ;
      A(    ;
      O     DB42.DBX  381.0;
      O     DB42.DBX  381.1;
      )     ;
      FP    M     20.0;
      =     L      2.0;
      A     L      2.0;
      JNB   _065;
      L     DB42.DBW  316;
      L     DB42.DBW  220;
      +I    ;
      T     DB42.DBW  316;
_065: NOP   0;
      A     L      2.0;
      JNB   _066;
      L     DB42.DBW  316;
      L     DB42.DBW  224;
      +I    ;
      T     DB42.DBW  316;
_066: NOP   0;
      A     L      2.0;
      JNB   _067;
      L     DB42.DBW  316;
      L     DB42.DBW  228;
      +I    ;
      T     DB42.DBW  316;
_067: NOP   0;
NETWORK
TITLE =용접누락버퍼로 공정DATA 전송1

      A(    ;
      O     M    164.1;
      O     M    164.0;
      )     ;
      A     M   1001.4;
      A     M   1001.5;
      A     M   1001.6;
      A(    ;
      O     DB42.DBX  380.0;
      O     DB42.DBX  380.1;
      )     ;
      A(    ;
      O     DB42.DBX  380.4;
      O     DB42.DBX  380.5;
      )     ;
      A(    ;
      O     DB42.DBX  381.0;
      O     DB42.DBX  381.1;
      )     ;
      FP    M     20.1;
      =     L      2.0;
      A     L      2.0;
      JNB   _068;
      CALL SFC   20 (
           SRCBLK                   := P#DB42.DBX 200.0 WORD 60,
           RET_VAL                  := #SFC20_RET_VAL,
           DSTBLK                   := P#DB43.DBX 1200.0 WORD 60);
_068: NOP   0;
      A     L      2.0;
      JNB   _069;
      CALL SFC   20 (
           SRCBLK                   := P#M 160.0 WORD 10,
           RET_VAL                  := #SFC20_RET_VAL,
           DSTBLK                   := P#DB45.DBX 200.0 WORD 10);
_069: NOP   0;
NETWORK
TITLE =

      A     M   4108.2;
      FP    M     20.2;
      =     L      2.0;
      A(    ;
      A     L      2.0;
      JNB   _06a;
      CALL SFC   20 (
           SRCBLK                   := P#DB43.DBX 2160.0 WORD 60,
           RET_VAL                  := #SFC20_RET_VAL,
           DSTBLK                   := P#DB43.DBX 2280.0 WORD 60);
_06a: A     BR;
      )     ;
      JNB   _06b;
      CALL SFC   20 (
           SRCBLK                   := P#DB43.DBX 2040.0 WORD 60,
           RET_VAL                  := #SFC20_RET_VAL,
           DSTBLK                   := P#DB43.DBX 2160.0 WORD 60);
_06b: NOP   0;
      A(    ;
      A     L      2.0;
      JNB   _06c;
      CALL SFC   20 (
           SRCBLK                   := P#DB43.DBX 1920.0 WORD 60,
           RET_VAL                  := #SFC20_RET_VAL,
           DSTBLK                   := P#DB43.DBX 2040.0 WORD 60);
_06c: A     BR;
      )     ;
      JNB   _06d;
      CALL SFC   20 (
           SRCBLK                   := P#DB43.DBX 1800.0 WORD 60,
           RET_VAL                  := #SFC20_RET_VAL,
           DSTBLK                   := P#DB43.DBX 1920.0 WORD 60);
_06d: NOP   0;
      A(    ;
      A     L      2.0;
      JNB   _06e;
      CALL SFC   20 (
           SRCBLK                   := P#DB43.DBX 1680.0 WORD 60,
           RET_VAL                  := #SFC20_RET_VAL,
           DSTBLK                   := P#DB43.DBX 1800.0 WORD 60);
_06e: A     BR;
      )     ;
      JNB   _06f;
      CALL SFC   20 (
           SRCBLK                   := P#DB43.DBX 1560.0 WORD 60,
           RET_VAL                  := #SFC20_RET_VAL,
           DSTBLK                   := P#DB43.DBX 1680.0 WORD 60);
_06f: NOP   0;
      A(    ;
      A     L      2.0;
      JNB   _070;
      CALL SFC   20 (
           SRCBLK                   := P#DB43.DBX 1440.0 WORD 60,
           RET_VAL                  := #SFC20_RET_VAL,
           DSTBLK                   := P#DB43.DBX 1560.0 WORD 60);
_070: A     BR;
      )     ;
      JNB   _071;
      CALL SFC   20 (
           SRCBLK                   := P#DB43.DBX 1320.0 WORD 60,
           RET_VAL                  := #SFC20_RET_VAL,
           DSTBLK                   := P#DB43.DBX 1440.0 WORD 60);
_071: NOP   0;
      A     L      2.0;
      JNB   _072;
      CALL SFC   20 (
           SRCBLK                   := P#DB43.DBX 1200.0 WORD 60,
           RET_VAL                  := #SFC20_RET_VAL,
           DSTBLK                   := P#DB43.DBX 1320.0 WORD 60);
_072: NOP   0;
      A     L      2.0;
      JNB   _073;
      CALL SFC   21 (
           IN0                      := P#M 40.0 WORD 1,
           RET_VAL                  := #SFC20_RET_VAL,
           OUT1                     := P#DB43.DBX 1200.0 WORD 60);
_073: NOP   0;
      A(    ;
      A     L      2.0;
      JNB   _074;
      CALL SFC   20 (
           SRCBLK                   := P#DB45.DBX 360.0 WORD 10,
           RET_VAL                  := #SFC20_RET_VAL,
           DSTBLK                   := P#DB45.DBX 380.0 WORD 10);
_074: A     BR;
      )     ;
      JNB   _075;
      CALL SFC   20 (
           SRCBLK                   := P#DB45.DBX 340.0 WORD 10,
           RET_VAL                  := #SFC20_RET_VAL,
           DSTBLK                   := P#DB45.DBX 360.0 WORD 10);
_075: NOP   0;
      A(    ;
      A     L      2.0;
      JNB   _076;
      CALL SFC   20 (
           SRCBLK                   := P#DB45.DBX 320.0 WORD 10,
           RET_VAL                  := #SFC20_RET_VAL,
           DSTBLK                   := P#DB45.DBX 340.0 WORD 10);
_076: A     BR;
      )     ;
      JNB   _077;
      CALL SFC   20 (
           SRCBLK                   := P#DB45.DBX 300.0 WORD 10,
           RET_VAL                  := #SFC20_RET_VAL,
           DSTBLK                   := P#DB45.DBX 320.0 WORD 10);
_077: NOP   0;
      A(    ;
      A     L      2.0;
      JNB   _078;
      CALL SFC   20 (
           SRCBLK                   := P#DB45.DBX 280.0 WORD 10,
           RET_VAL                  := #SFC20_RET_VAL,
           DSTBLK                   := P#DB45.DBX 300.0 WORD 10);
_078: A     BR;
      )     ;
      JNB   _079;
      CALL SFC   20 (
           SRCBLK                   := P#DB45.DBX 260.0 WORD 10,
           RET_VAL                  := #SFC20_RET_VAL,
           DSTBLK                   := P#DB45.DBX 280.0 WORD 10);
_079: NOP   0;
      A(    ;
      A     L      2.0;
      JNB   _07a;
      CALL SFC   20 (
           SRCBLK                   := P#DB45.DBX 240.0 WORD 10,
           RET_VAL                  := #SFC20_RET_VAL,
           DSTBLK                   := P#DB45.DBX 260.0 WORD 10);
_07a: A     BR;
      )     ;
      JNB   _07b;
      CALL SFC   20 (
           SRCBLK                   := P#DB45.DBX 220.0 WORD 10,
           RET_VAL                  := #SFC20_RET_VAL,
           DSTBLK                   := P#DB45.DBX 240.0 WORD 10);
_07b: NOP   0;
      A     L      2.0;
      JNB   _07c;
      CALL SFC   20 (
           SRCBLK                   := P#DB45.DBX 200.0 WORD 10,
           RET_VAL                  := #SFC20_RET_VAL,
           DSTBLK                   := P#DB45.DBX 220.0 WORD 10);
_07c: NOP   0;
      A     L      2.0;
      JNB   _07d;
      CALL SFC   21 (
           IN0                      := P#M 40.0 WORD 1,
           RET_VAL                  := #SFC20_RET_VAL,
           OUT1                     := P#DB45.DBX 200.0 WORD 10);
_07d: NOP   0;
NETWORK
TITLE =용접누락버퍼로 공정DATA 전송1
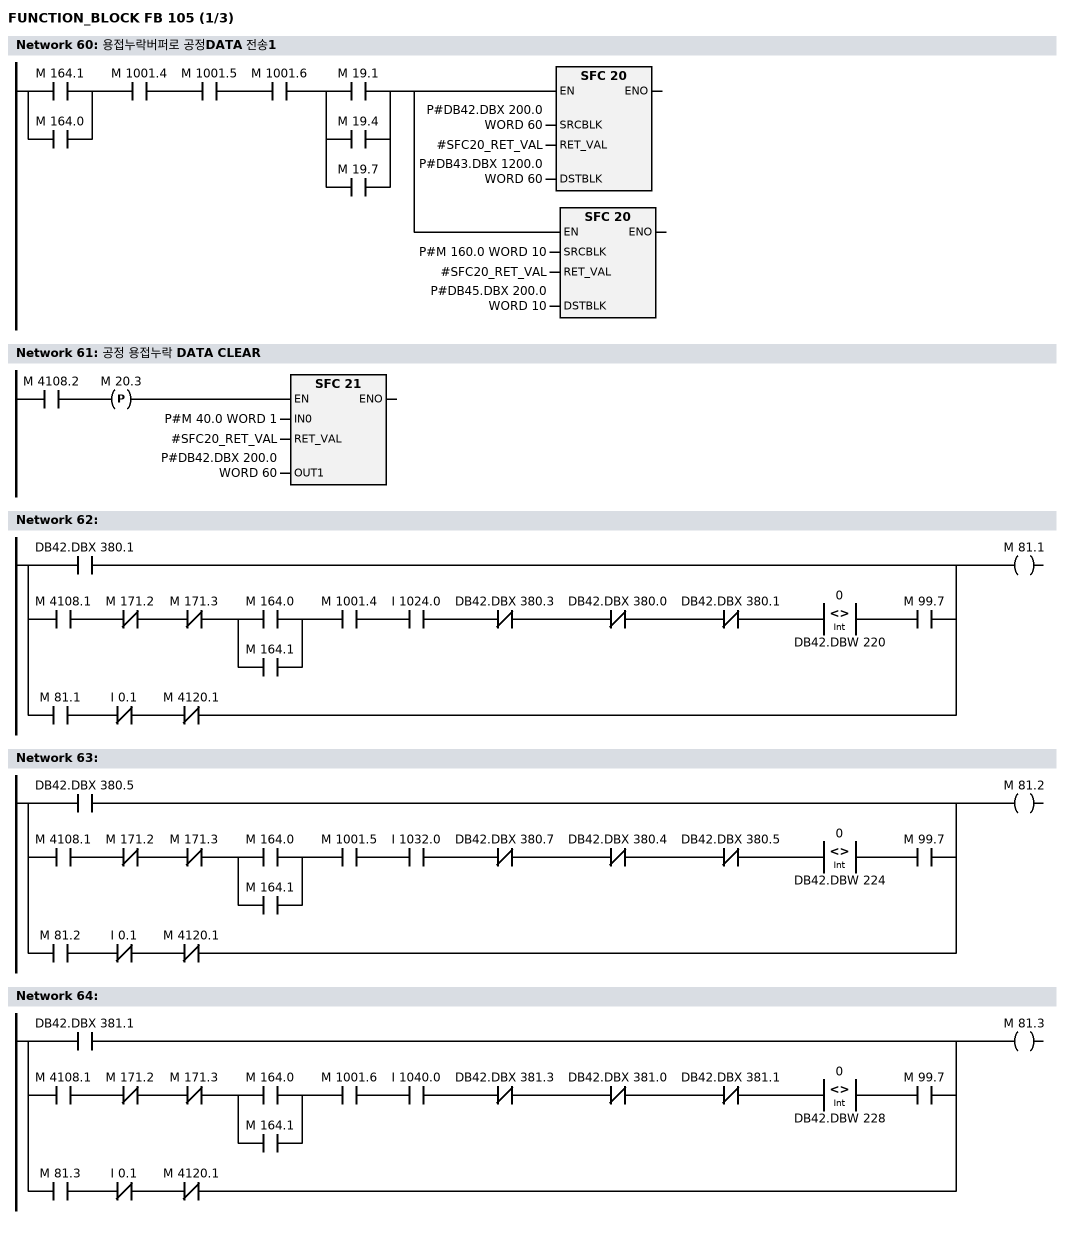

      A(    ;
      O     M    164.1;
      O     M    164.0;
      )     ;
      A     M   1001.4;
      A     M   1001.5;
      A     M   1001.6;
      A(    ;
      O     M     19.1;
      O     M     19.4;
      O     M     19.7;
      )     ;
      =     L      2.0;
      A     L      2.0;
      JNB   _07e;
      CALL SFC   20 (
           SRCBLK                   := P#DB42.DBX 200.0 WORD 60,
           RET_VAL                  := #SFC20_RET_VAL,
           DSTBLK                   := P#DB43.DBX 1200.0 WORD 60);
_07e: NOP   0;
      A     L      2.0;
      JNB   _07f;
      CALL SFC   20 (
           SRCBLK                   := P#M 160.0 WORD 10,
           RET_VAL                  := #SFC20_RET_VAL,
           DSTBLK                   := P#DB45.DBX 200.0 WORD 10);
_07f: NOP   0;
NETWORK
TITLE =공정 용접누락 DATA CLEAR

      A     M   4108.2;
      FP    M     20.3;
      JNB   _080;
      CALL SFC   21 (
           IN0                      := P#M 40.0 WORD 1,
           RET_VAL                  := #SFC20_RET_VAL,
           OUT1                     := P#DB42.DBX 200.0 WORD 60);
_080: NOP   0;
NETWORK
TITLE =

      O     DB42.DBX  380.1;
      O     ;
      A     M   4108.1;
      AN    M    171.2;
      AN    M    171.3;
      A(    ;
      O     M    164.0;
      O     M    164.1;
      )     ;
      A     M   1001.4;
      A     I   1024.0;
      AN    DB42.DBX  380.3;
      AN    DB42.DBX  380.0;
      AN    DB42.DBX  380.1;
      A(    ;
      L     0;
      L     DB42.DBW  220;
      <>I   ;
      )     ;
      A     M     99.7;
      O     ;
      A     M     81.1;
      AN    I      0.1;
      AN    M   4120.1;
      =     M     81.1;
NETWORK
TITLE =

      O     DB42.DBX  380.5;
      O     ;
      A     M   4108.1;
      AN    M    171.2;
      AN    M    171.3;
      A(    ;
      O     M    164.0;
      O     M    164.1;
      )     ;
      A     M   1001.5;
      A     I   1032.0;
      AN    DB42.DBX  380.7;
      AN    DB42.DBX  380.4;
      AN    DB42.DBX  380.5;
      A(    ;
      L     0;
      L     DB42.DBW  224;
      <>I   ;
      )     ;
      A     M     99.7;
      O     ;
      A     M     81.2;
      AN    I      0.1;
      AN    M   4120.1;
      =     M     81.2;
NETWORK
TITLE =

      O     DB42.DBX  381.1;
      O     ;
      A     M   4108.1;
      AN    M    171.2;
      AN    M    171.3;
      A(    ;
      O     M    164.0;
      O     M    164.1;
      )     ;
      A     M   1001.6;
      A     I   1040.0;
      AN    DB42.DBX  381.3;
      AN    DB42.DBX  381.0;
      AN    DB42.DBX  381.1;
      A(    ;
      L     0;
      L     DB42.DBW  228;
      <>I   ;
      )     ;
      A     M     99.7;
      O     ;
      A     M     81.3;
      AN    I      0.1;
      AN    M   4120.1;
      =     M     81.3;
NETWORK
TITLE =
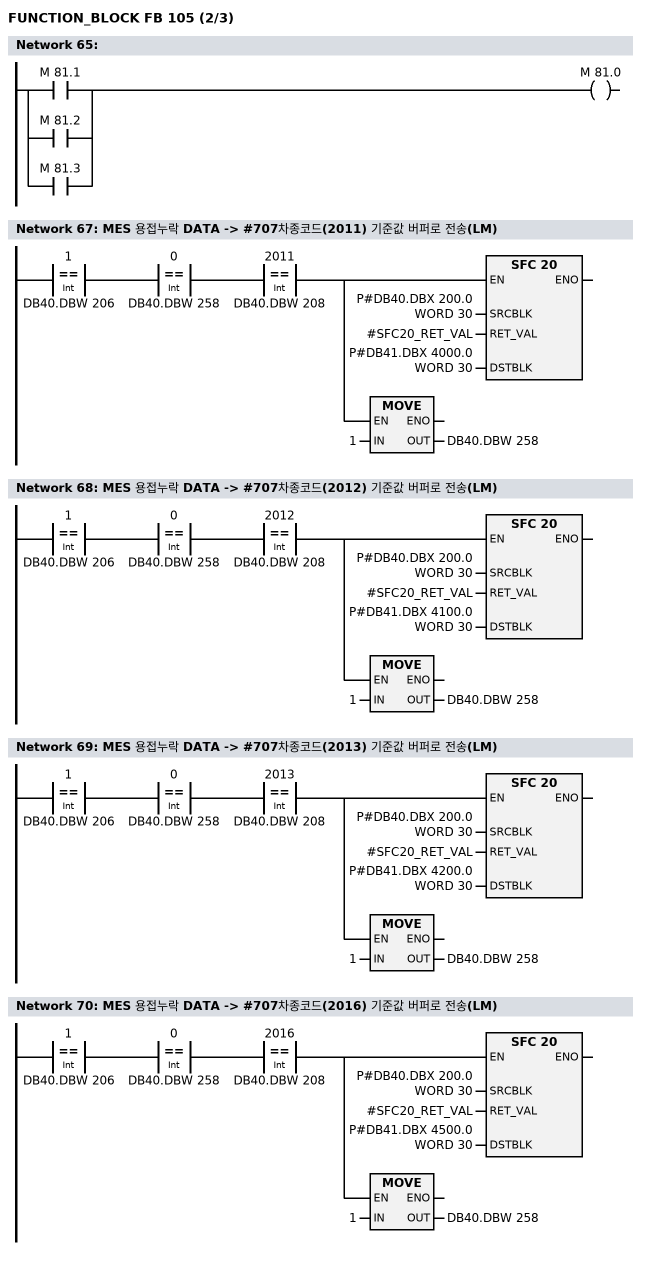

      O     M     81.1;
      O     M     81.2;
      O     M     81.3;
      =     M     81.0;
NETWORK
TITLE =

NETWORK
TITLE =MES 용접누락 DATA -> #707차종코드(2011) 기준값 버퍼로 전송(LM)

      A(    ;
      L     1;
      L     DB40.DBW  206;
      ==I   ;
      )     ;
      A(    ;
      L     0;
      L     DB40.DBW  258;
      ==I   ;
      )     ;
      A(    ;
      L     2011;
      L     DB40.DBW  208;
      ==I   ;
      )     ;
      =     L      2.0;
      A     L      2.0;
      JNB   _081;
      CALL SFC   20 (
           SRCBLK                   := P#DB40.DBX 200.0 WORD 30,
           RET_VAL                  := #SFC20_RET_VAL,
           DSTBLK                   := P#DB41.DBX 4000.0 WORD 30);
_081: NOP   0;
      A     L      2.0;
      JNB   _082;
      L     1;
      T     DB40.DBW  258;
_082: NOP   0;
NETWORK
TITLE =MES 용접누락 DATA -> #707차종코드(2012) 기준값 버퍼로 전송(LM)

      A(    ;
      L     1;
      L     DB40.DBW  206;
      ==I   ;
      )     ;
      A(    ;
      L     0;
      L     DB40.DBW  258;
      ==I   ;
      )     ;
      A(    ;
      L     2012;
      L     DB40.DBW  208;
      ==I   ;
      )     ;
      =     L      2.0;
      A     L      2.0;
      JNB   _083;
      CALL SFC   20 (
           SRCBLK                   := P#DB40.DBX 200.0 WORD 30,
           RET_VAL                  := #SFC20_RET_VAL,
           DSTBLK                   := P#DB41.DBX 4100.0 WORD 30);
_083: NOP   0;
      A     L      2.0;
      JNB   _084;
      L     1;
      T     DB40.DBW  258;
_084: NOP   0;
NETWORK
TITLE =MES 용접누락 DATA -> #707차종코드(2013) 기준값 버퍼로 전송(LM)
//
//
      A(    ;
      L     1;
      L     DB40.DBW  206;
      ==I   ;
      )     ;
      A(    ;
      L     0;
      L     DB40.DBW  258;
      ==I   ;
      )     ;
      A(    ;
      L     2013;
      L     DB40.DBW  208;
      ==I   ;
      )     ;
      =     L      2.0;
      A     L      2.0;
      JNB   _085;
      CALL SFC   20 (
           SRCBLK                   := P#DB40.DBX 200.0 WORD 30,
           RET_VAL                  := #SFC20_RET_VAL,
           DSTBLK                   := P#DB41.DBX 4200.0 WORD 30);
_085: NOP   0;
      A     L      2.0;
      JNB   _086;
      L     1;
      T     DB40.DBW  258;
_086: NOP   0;
NETWORK
TITLE =MES 용접누락 DATA -> #707차종코드(2016) 기준값 버퍼로 전송(LM)

      A(    ;
      L     1;
      L     DB40.DBW  206;
      ==I   ;
      )     ;
      A(    ;
      L     0;
      L     DB40.DBW  258;
      ==I   ;
      )     ;
      A(    ;
      L     2016;
      L     DB40.DBW  208;
      ==I   ;
      )     ;
      =     L      2.0;
      A     L      2.0;
      JNB   _087;
      CALL SFC   20 (
           SRCBLK                   := P#DB40.DBX 200.0 WORD 30,
           RET_VAL                  := #SFC20_RET_VAL,
           DSTBLK                   := P#DB41.DBX 4500.0 WORD 30);
_087: NOP   0;
      A     L      2.0;
      JNB   _088;
      L     1;
      T     DB40.DBW  258;
_088: NOP   0;
NETWORK
TITLE =MES 용접누락 DATA -> #707차종코드(2017) 기준값 버퍼로 전송(LM)
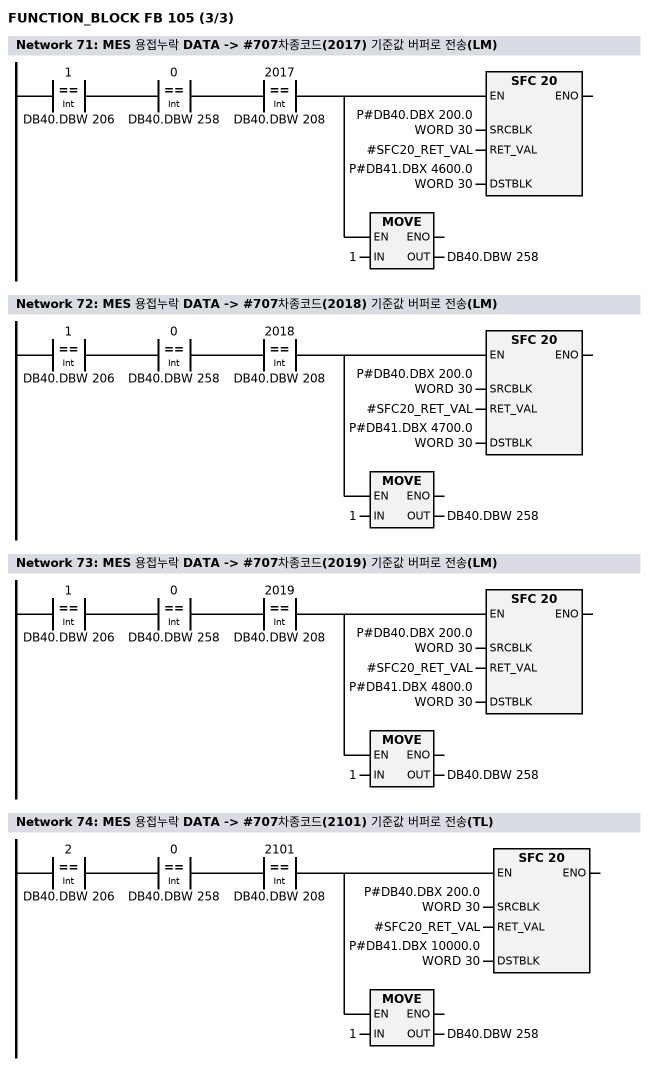

      A(    ;
      L     1;
      L     DB40.DBW  206;
      ==I   ;
      )     ;
      A(    ;
      L     0;
      L     DB40.DBW  258;
      ==I   ;
      )     ;
      A(    ;
      L     2017;
      L     DB40.DBW  208;
      ==I   ;
      )     ;
      =     L      2.0;
      A     L      2.0;
      JNB   _089;
      CALL SFC   20 (
           SRCBLK                   := P#DB40.DBX 200.0 WORD 30,
           RET_VAL                  := #SFC20_RET_VAL,
           DSTBLK                   := P#DB41.DBX 4600.0 WORD 30);
_089: NOP   0;
      A     L      2.0;
      JNB   _08a;
      L     1;
      T     DB40.DBW  258;
_08a: NOP   0;
NETWORK
TITLE =MES 용접누락 DATA -> #707차종코드(2018) 기준값 버퍼로 전송(LM)

      A(    ;
      L     1;
      L     DB40.DBW  206;
      ==I   ;
      )     ;
      A(    ;
      L     0;
      L     DB40.DBW  258;
      ==I   ;
      )     ;
      A(    ;
      L     2018;
      L     DB40.DBW  208;
      ==I   ;
      )     ;
      =     L      2.0;
      A     L      2.0;
      JNB   _08b;
      CALL SFC   20 (
           SRCBLK                   := P#DB40.DBX 200.0 WORD 30,
           RET_VAL                  := #SFC20_RET_VAL,
           DSTBLK                   := P#DB41.DBX 4700.0 WORD 30);
_08b: NOP   0;
      A     L      2.0;
      JNB   _08c;
      L     1;
      T     DB40.DBW  258;
_08c: NOP   0;
NETWORK
TITLE =MES 용접누락 DATA -> #707차종코드(2019) 기준값 버퍼로 전송(LM)

      A(    ;
      L     1;
      L     DB40.DBW  206;
      ==I   ;
      )     ;
      A(    ;
      L     0;
      L     DB40.DBW  258;
      ==I   ;
      )     ;
      A(    ;
      L     2019;
      L     DB40.DBW  208;
      ==I   ;
      )     ;
      =     L      2.0;
      A     L      2.0;
      JNB   _08d;
      CALL SFC   20 (
           SRCBLK                   := P#DB40.DBX 200.0 WORD 30,
           RET_VAL                  := #SFC20_RET_VAL,
           DSTBLK                   := P#DB41.DBX 4800.0 WORD 30);
_08d: NOP   0;
      A     L      2.0;
      JNB   _08e;
      L     1;
      T     DB40.DBW  258;
_08e: NOP   0;
NETWORK
TITLE =MES 용접누락 DATA -> #707차종코드(2101) 기준값 버퍼로 전송(TL)

      A(    ;
      L     2;
      L     DB40.DBW  206;
      ==I   ;
      )     ;
      A(    ;
      L     0;
      L     DB40.DBW  258;
      ==I   ;
      )     ;
      A(    ;
      L     2101;
      L     DB40.DBW  208;
      ==I   ;
      )     ;
      =     L      2.0;
      A     L      2.0;
      JNB   _08f;
      CALL SFC   20 (
           SRCBLK                   := P#DB40.DBX 200.0 WORD 30,
           RET_VAL                  := #SFC20_RET_VAL,
           DSTBLK                   := P#DB41.DBX 10000.0 WORD 30);
_08f: NOP   0;
      A     L      2.0;
      JNB   _090;
      L     1;
      T     DB40.DBW  258;
_090: NOP   0;
NETWORK
TITLE =#707 RBT1호 용접카운터 INT -> DB로 전송보조

      AN    OV;
      =     L      2.0;
      A     L      2.0;
      A     I   1052.0;
      =     M     21.0;
      A     L      2.0;
      A     I   1052.1;
      =     M     21.1;
      A     L      2.0;
      A     I   1052.2;
      =     M     21.2;
      A     L      2.0;
      A     I   1052.3;
      =     M     21.3;
      A     L      2.0;
      A     I   1052.4;
      =     M     21.4;
      A     L      2.0;
      AN    M      3.3;
      =     L      2.1;
      A     L      2.1;
      A     I   1052.5;
      =     M     21.5;
      A     L      2.1;
      A     I   1052.6;
      =     M     21.6;
      A     L      2.1;
      A     I   1052.7;
      =     M     21.7;
NETWORK
TITLE =#707 RBT1호 용접카운터 INT -> DB로 전송
//
//
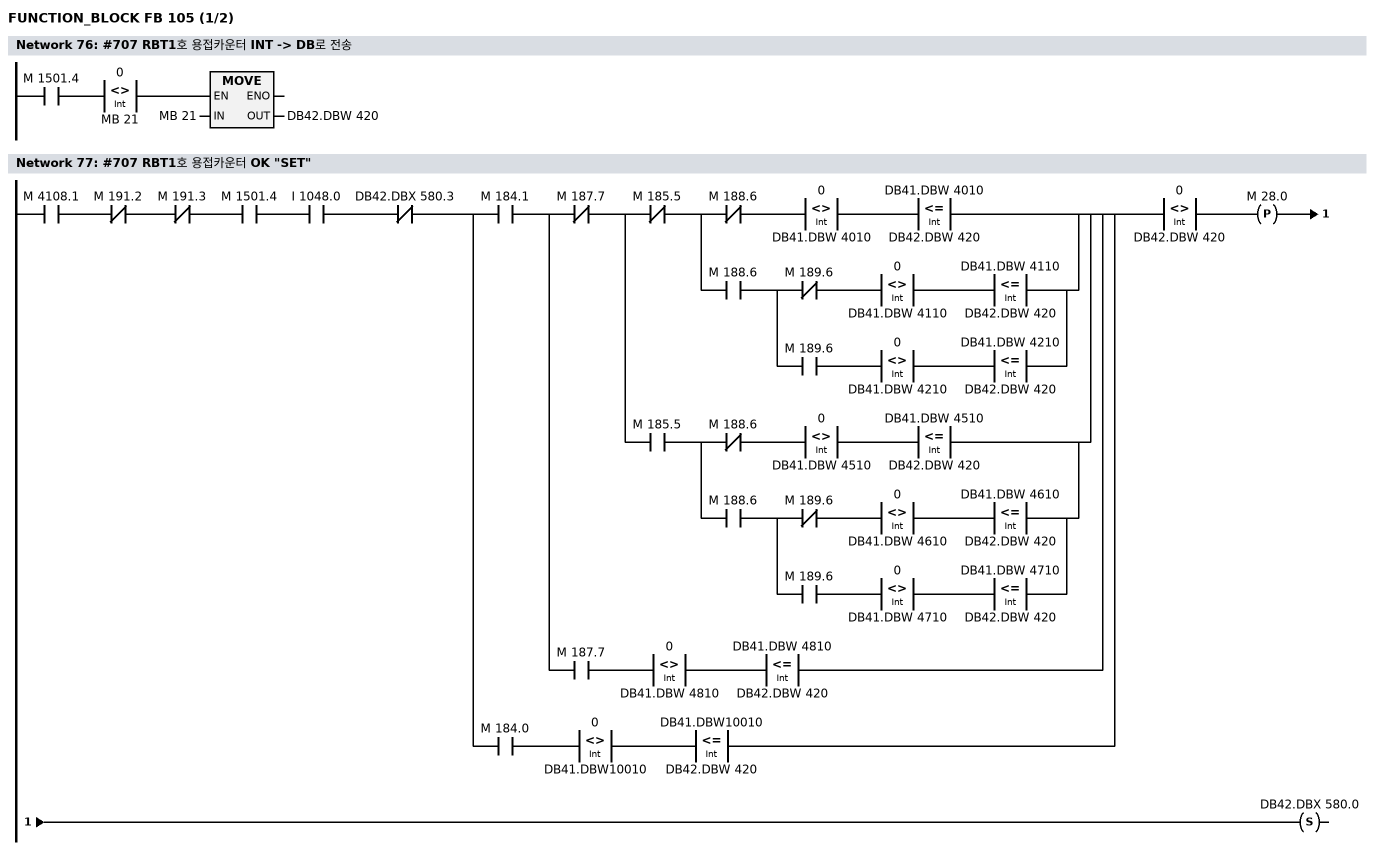
      A     M   1501.4;
      A(    ;
      L     0;
      L     MB    21;
      <>I   ;
      )     ;
      JNB   _091;
      L     MB    21;
      T     DB42.DBW  420;
_091: NOP   0;
NETWORK
TITLE =#707 RBT1호 용접카운터 OK "SET"

      A     M   4108.1;
      AN    M    191.2;
      AN    M    191.3;
      A     M   1501.4;
      A     I   1048.0;
      AN    DB42.DBX  580.3;
      A(    ;
      A     M    184.1;
      A(    ;
      AN    M    187.7;
      A(    ;
      AN    M    185.5;
      A(    ;
      AN    M    188.6;
      A(    ;
      L     0;
      L     DB41.DBW 4010;
      <>I   ;
      )     ;
      A(    ;
      L     DB41.DBW 4010;
      L     DB42.DBW  420;
      <=I   ;
      )     ;
      O     ;
      A     M    188.6;
      A(    ;
      AN    M    189.6;
      A(    ;
      L     0;
      L     DB41.DBW 4110;
      <>I   ;
      )     ;
      A(    ;
      L     DB41.DBW 4110;
      L     DB42.DBW  420;
      <=I   ;
      )     ;
      O     ;
      A     M    189.6;
      A(    ;
      L     0;
      L     DB41.DBW 4210;
      <>I   ;
      )     ;
      A(    ;
      L     DB41.DBW 4210;
      L     DB42.DBW  420;
      <=I   ;
      )     ;
      )     ;
      )     ;
      O     ;
      A     M    185.5;
      A(    ;
      AN    M    188.6;
      A(    ;
      L     0;
      L     DB41.DBW 4510;
      <>I   ;
      )     ;
      A(    ;
      L     DB41.DBW 4510;
      L     DB42.DBW  420;
      <=I   ;
      )     ;
      O     ;
      A     M    188.6;
      A(    ;
      AN    M    189.6;
      A(    ;
      L     0;
      L     DB41.DBW 4610;
      <>I   ;
      )     ;
      A(    ;
      L     DB41.DBW 4610;
      L     DB42.DBW  420;
      <=I   ;
      )     ;
      O     ;
      A     M    189.6;
      A(    ;
      L     0;
      L     DB41.DBW 4710;
      <>I   ;
      )     ;
      A(    ;
      L     DB41.DBW 4710;
      L     DB42.DBW  420;
      <=I   ;
      )     ;
      )     ;
      )     ;
      )     ;
      O     ;
      A     M    187.7;
      A(    ;
      L     0;
      L     DB41.DBW 4810;
      <>I   ;
      )     ;
      A(    ;
      L     DB41.DBW 4810;
      L     DB42.DBW  420;
      <=I   ;
      )     ;
      )     ;
      O     ;
      A     M    184.0;
      A(    ;
      L     0;
      L     DB41.DBW10010;
      <>I   ;
      )     ;
      A(    ;
      L     DB41.DBW10010;
      L     DB42.DBW  420;
      <=I   ;
      )     ;
      )     ;
      A(    ;
      L     0;
      L     DB42.DBW  420;
      <>I   ;
      )     ;
      FP    M     28.0;
      S     DB42.DBX  580.0;
NETWORK
TITLE =#707 RBT1호 용접카운터 NG "SET"
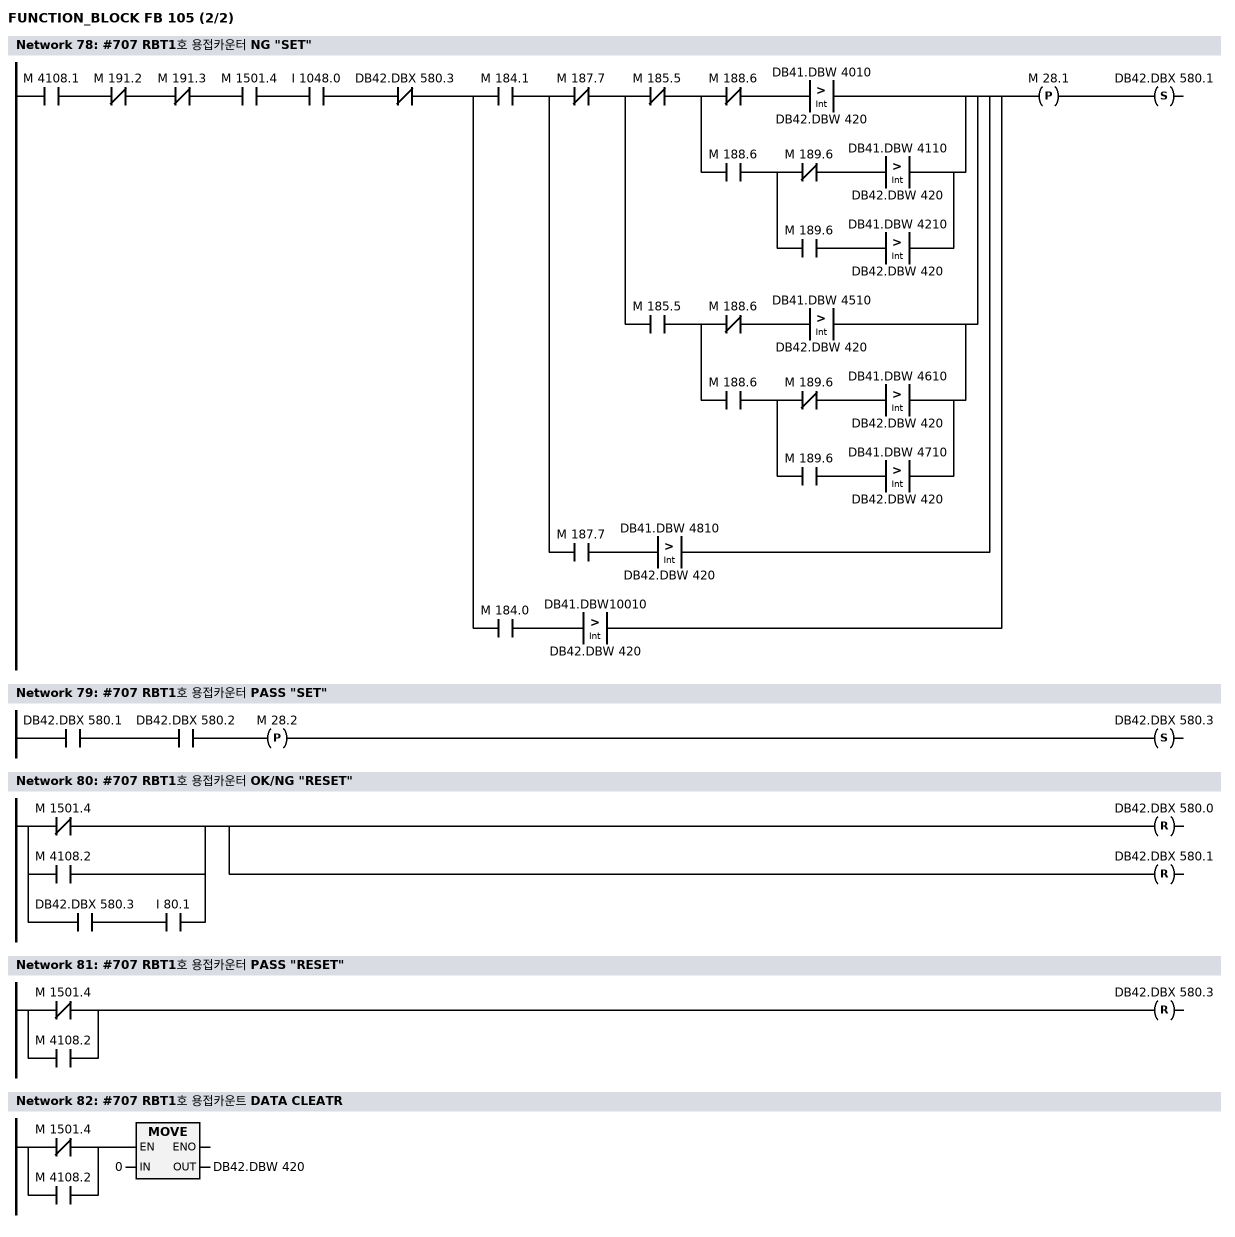

      A     M   4108.1;
      AN    M    191.2;
      AN    M    191.3;
      A     M   1501.4;
      A     I   1048.0;
      AN    DB42.DBX  580.3;
      A(    ;
      A     M    184.1;
      A(    ;
      AN    M    187.7;
      A(    ;
      AN    M    185.5;
      A(    ;
      AN    M    188.6;
      A(    ;
      L     DB41.DBW 4010;
      L     DB42.DBW  420;
      >I    ;
      )     ;
      O     ;
      A     M    188.6;
      A(    ;
      AN    M    189.6;
      A(    ;
      L     DB41.DBW 4110;
      L     DB42.DBW  420;
      >I    ;
      )     ;
      O     ;
      A     M    189.6;
      A(    ;
      L     DB41.DBW 4210;
      L     DB42.DBW  420;
      >I    ;
      )     ;
      )     ;
      )     ;
      O     ;
      A     M    185.5;
      A(    ;
      AN    M    188.6;
      A(    ;
      L     DB41.DBW 4510;
      L     DB42.DBW  420;
      >I    ;
      )     ;
      O     ;
      A     M    188.6;
      A(    ;
      AN    M    189.6;
      A(    ;
      L     DB41.DBW 4610;
      L     DB42.DBW  420;
      >I    ;
      )     ;
      O     ;
      A     M    189.6;
      A(    ;
      L     DB41.DBW 4710;
      L     DB42.DBW  420;
      >I    ;
      )     ;
      )     ;
      )     ;
      )     ;
      O     ;
      A     M    187.7;
      A(    ;
      L     DB41.DBW 4810;
      L     DB42.DBW  420;
      >I    ;
      )     ;
      )     ;
      O     ;
      A     M    184.0;
      A(    ;
      L     DB41.DBW10010;
      L     DB42.DBW  420;
      >I    ;
      )     ;
      )     ;
      FP    M     28.1;
      S     DB42.DBX  580.1;
NETWORK
TITLE =#707 RBT1호 용접카운터 PASS "SET"

      A     DB42.DBX  580.1;
      A     DB42.DBX  580.2;
      FP    M     28.2;
      S     DB42.DBX  580.3;
NETWORK
TITLE =#707 RBT1호 용접카운터 OK/NG "RESET"

      ON    M   1501.4;
      O     M   4108.2;
      O     ;
      A     DB42.DBX  580.3;
      A     I     80.1;
      R     DB42.DBX  580.0;
      R     DB42.DBX  580.1;
NETWORK
TITLE =#707 RBT1호 용접카운터 PASS "RESET"

      ON    M   1501.4;
      O     M   4108.2;
      R     DB42.DBX  580.3;
NETWORK
TITLE =#707 RBT1호 용접카운트 DATA CLEATR

      A(    ;
      ON    M   1501.4;
      O     M   4108.2;
      )     ;
      JNB   _092;
      L     0;
      T     DB42.DBW  420;
_092: NOP   0;
NETWORK
TITLE =#707 RBT2호 용접카운터 INT -> DB로 전송보조

      AN    OV;
      =     L      2.0;
      A     L      2.0;
      A     I   1060.0;
      =     M     22.0;
      A     L      2.0;
      A     I   1060.1;
      =     M     22.1;
      A     L      2.0;
      A     I   1060.2;
      =     M     22.2;
      A     L      2.0;
      A     I   1060.3;
      =     M     22.3;
      A     L      2.0;
      A     I   1060.4;
      =     M     22.4;
      A     L      2.0;
      AN    M      3.3;
      =     L      2.1;
      A     L      2.1;
      A     I   1060.5;
      =     M     22.5;
      A     L      2.1;
      A     I   1060.6;
      =     M     22.6;
      A     L      2.1;
      A     I   1060.7;
      =     M     22.7;
NETWORK
TITLE =#707 RBT2호 용접카운터 INT -> DB로 전송
